Fanuc TP program (LS listing): CODE3.ls

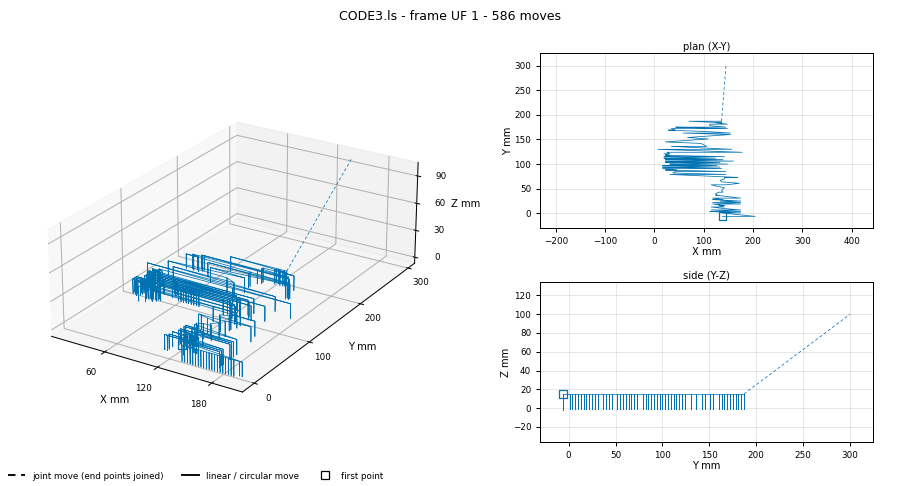
[picture p0: tool path of CODE3.ls in frame UF 1, 586 of 586 moves have a stored position in this frame; points joined in program order, loops and branches not executed]
/PROG CODE3
/ATTR
OWNER		= NOC_FANU;
COMMENT		= "NOC_FANUC";
PROG_SIZE	= 328;
CREATE		= DATE 97-07-08  TIME 03:05:20;
MODIFIED	= DATE 17-07-08  TIME 03:05:26;
FILE_NAME	= ;
VERSION		= 0;
LINE_COUNT	= 10;
MEMORY_SIZE	= 692;
PROTECT		= READ_WRITE;
TCD:  STACK_SIZE	= 0,
      TASK_PRIORITY	= 0,
      TIME_SLICE	= 0,
      BUSY_LAMP_OFF	= 0,
      ABORT_REQUEST	= 0,
      PAUSE_REQUEST	= 0;
DEFAULT_GROUP	= 1,*,*,*,*;
CONTROL_CODE	= 00000000 00000000;
/APPL
/MN
1:UFRAME_NUM=1 ;
2:UTOOL_NUM=3;
3:J P[133] 10% CNT100;
4:L P[134] 250mm/sec FINE;
5:L P[135] 250mm/sec CNT100;
6:L P[136] 250mm/sec CNT100;
7:L P[137] 250mm/sec FINE;
8:L P[138] 250mm/sec CNT100;
9:L P[139] 250mm/sec CNT100;
10:L P[140] 250mm/sec FINE;
11:L P[141] 250mm/sec CNT100;
12:L P[142] 250mm/sec CNT100;
13:L P[143] 250mm/sec FINE;
14:L P[144] 250mm/sec CNT100;
15:L P[145] 250mm/sec CNT100;
16:L P[146] 250mm/sec FINE;
17:L P[147] 250mm/sec CNT100;
18:L P[148] 250mm/sec CNT100;
19:L P[149] 250mm/sec FINE;
20:L P[150] 250mm/sec CNT100;
21:L P[151] 250mm/sec CNT100;
22:L P[152] 250mm/sec FINE;
23:L P[153] 250mm/sec CNT100;
24:L P[154] 250mm/sec CNT100;
25:L P[155] 250mm/sec FINE;
26:L P[156] 250mm/sec CNT100;
27:L P[157] 250mm/sec CNT100;
28:L P[158] 250mm/sec FINE;
29:L P[159] 250mm/sec CNT100;
30:L P[160] 250mm/sec CNT100;
31:L P[161] 250mm/sec FINE;
32:L P[162] 250mm/sec CNT100;
33:L P[163] 250mm/sec CNT100;
34:L P[164] 250mm/sec FINE;
35:L P[165] 250mm/sec CNT100;
36:L P[166] 250mm/sec CNT100;
37:L P[167] 250mm/sec FINE;
38:L P[168] 250mm/sec CNT100;
39:L P[169] 250mm/sec CNT100;
40:L P[170] 250mm/sec FINE;
41:L P[171] 250mm/sec CNT100;
42:L P[172] 250mm/sec CNT100;
43:L P[173] 250mm/sec FINE;
44:L P[174] 250mm/sec CNT100;
45:L P[175] 250mm/sec CNT100;
46:L P[176] 250mm/sec FINE;
47:L P[177] 250mm/sec CNT100;
48:L P[178] 250mm/sec CNT100;
49:L P[179] 250mm/sec FINE;
50:L P[180] 250mm/sec CNT100;
51:L P[181] 250mm/sec CNT100;
52:L P[182] 250mm/sec FINE;
53:L P[183] 250mm/sec CNT100;
54:L P[184] 250mm/sec CNT100;
55:L P[185] 250mm/sec FINE;
56:L P[186] 250mm/sec CNT100;
57:L P[187] 250mm/sec CNT100;
58:L P[188] 250mm/sec FINE;
59:L P[189] 250mm/sec CNT100;
60:L P[190] 250mm/sec CNT100;
61:L P[191] 250mm/sec FINE;
62:L P[192] 250mm/sec CNT100;
63:L P[193] 250mm/sec CNT100;
64:L P[194] 250mm/sec FINE;
65:L P[195] 250mm/sec CNT100;
66:L P[196] 250mm/sec CNT100;
67:L P[197] 250mm/sec FINE;
68:L P[198] 250mm/sec CNT100;
69:L P[532] 250mm/sec CNT100;
70:L P[533] 250mm/sec FINE;
71:L P[534] 250mm/sec CNT100;
72:L P[553] 250mm/sec CNT100;
73:L P[554] 250mm/sec FINE;
74:L P[555] 250mm/sec CNT100;
75:L P[670] 250mm/sec CNT100;
76:L P[671] 250mm/sec FINE;
77:L P[672] 250mm/sec CNT100;
78:L P[673] 250mm/sec CNT100;
79:L P[674] 250mm/sec FINE;
80:L P[675] 250mm/sec CNT100;
81:L P[691] 250mm/sec CNT100;
82:L P[692] 250mm/sec FINE;
83:L P[693] 250mm/sec CNT100;
84:L P[721] 250mm/sec CNT100;
85:L P[722] 250mm/sec FINE;
86:L P[723] 250mm/sec CNT100;
87:L P[841] 250mm/sec CNT100;
88:L P[842] 250mm/sec FINE;
89:L P[843] 250mm/sec CNT100;
90:L P[865] 250mm/sec CNT100;
91:L P[866] 250mm/sec FINE;
92:L P[867] 250mm/sec CNT100;
93:L P[880] 250mm/sec CNT100;
94:L P[881] 250mm/sec FINE;
95:L P[882] 250mm/sec CNT100;
96:L P[1024] 250mm/sec CNT100;
97:L P[1025] 250mm/sec FINE;
98:L P[1026] 250mm/sec CNT100;
99:L P[1162] 250mm/sec CNT100;
100:L P[1163] 250mm/sec FINE;
101:L P[1164] 250mm/sec CNT100;
102:L P[1186] 250mm/sec CNT100;
103:L P[1187] 250mm/sec FINE;
104:L P[1188] 250mm/sec CNT100;
105:L P[1189] 250mm/sec CNT100;
106:L P[1190] 250mm/sec FINE;
107:L P[1191] 250mm/sec CNT100;
108:L P[1333] 250mm/sec CNT100;
109:L P[1334] 250mm/sec FINE;
110:L P[1335] 250mm/sec CNT100;
111:L P[1336] 250mm/sec CNT100;
112:L P[1337] 250mm/sec FINE;
113:L P[1338] 250mm/sec CNT100;
114:L P[1339] 250mm/sec CNT100;
115:L P[1340] 250mm/sec FINE;
116:L P[1341] 250mm/sec CNT100;
117:L P[1345] 250mm/sec CNT100;
118:L P[1346] 250mm/sec FINE;
119:L P[1347] 250mm/sec CNT100;
120:L P[1477] 250mm/sec CNT100;
121:L P[1478] 250mm/sec FINE;
122:L P[1479] 250mm/sec CNT100;
123:L P[1480] 250mm/sec CNT100;
124:L P[1481] 250mm/sec FINE;
125:L P[1482] 250mm/sec CNT100;
126:L P[1489] 250mm/sec CNT100;
127:L P[1490] 250mm/sec FINE;
128:L P[1491] 250mm/sec CNT100;
129:L P[1492] 250mm/sec CNT100;
130:L P[1493] 250mm/sec FINE;
131:L P[1494] 250mm/sec CNT100;
132:L P[1507] 250mm/sec CNT100;
133:L P[1508] 250mm/sec FINE;
134:L P[1509] 250mm/sec CNT100;
135:L P[1627] 250mm/sec CNT100;
136:L P[1628] 250mm/sec FINE;
137:L P[1629] 250mm/sec CNT100;
138:L P[1633] 250mm/sec CNT100;
139:L P[1634] 250mm/sec FINE;
140:L P[1635] 250mm/sec CNT100;
141:L P[1654] 250mm/sec CNT100;
142:L P[1655] 250mm/sec FINE;
143:L P[1656] 250mm/sec CNT100;
144:L P[1789] 250mm/sec CNT100;
145:L P[1790] 250mm/sec FINE;
146:L P[1791] 250mm/sec CNT100;
147:L P[1798] 250mm/sec CNT100;
148:L P[1799] 250mm/sec FINE;
149:L P[1800] 250mm/sec CNT100;
150:L P[1918] 250mm/sec CNT100;
151:L P[1919] 250mm/sec FINE;
152:L P[1920] 250mm/sec CNT100;
153:L P[1927] 250mm/sec CNT100;
154:L P[1928] 250mm/sec FINE;
155:L P[1929] 250mm/sec CNT100;
156:L P[1930] 250mm/sec CNT100;
157:L P[1931] 250mm/sec FINE;
158:L P[1932] 250mm/sec CNT100;
159:L P[1939] 250mm/sec CNT100;
160:L P[1940] 250mm/sec FINE;
161:L P[1941] 250mm/sec CNT100;
162:L P[2065] 250mm/sec CNT100;
163:L P[2066] 250mm/sec FINE;
164:L P[2067] 250mm/sec CNT100;
165:L P[2095] 250mm/sec CNT100;
166:L P[2096] 250mm/sec FINE;
167:L P[2097] 250mm/sec CNT100;
168:L P[2371] 250mm/sec CNT100;
169:L P[2372] 250mm/sec FINE;
170:L P[2373] 250mm/sec CNT100;
171:L P[2374] 250mm/sec CNT100;
172:L P[2375] 250mm/sec FINE;
173:L P[2376] 250mm/sec CNT100;
174:L P[2512] 250mm/sec CNT100;
175:L P[2513] 250mm/sec FINE;
176:L P[2514] 250mm/sec CNT100;
177:L P[2656] 250mm/sec CNT100;
178:L P[2657] 250mm/sec FINE;
179:L P[2658] 250mm/sec CNT100;
180:L P[2665] 250mm/sec CNT100;
181:L P[2666] 250mm/sec FINE;
182:L P[2667] 250mm/sec CNT100;
183:L P[2803] 250mm/sec CNT100;
184:L P[2804] 250mm/sec FINE;
185:L P[2805] 250mm/sec CNT100;
186:L P[3121] 250mm/sec CNT100;
187:L P[3122] 250mm/sec FINE;
188:L P[3123] 250mm/sec CNT100;
189:L P[3256] 250mm/sec CNT100;
190:L P[3257] 250mm/sec FINE;
191:L P[3258] 250mm/sec CNT100;
192:L P[3394] 250mm/sec CNT100;
193:L P[3395] 250mm/sec FINE;
194:L P[3396] 250mm/sec CNT100;
195:L P[3397] 250mm/sec CNT100;
196:L P[3398] 250mm/sec FINE;
197:L P[3399] 250mm/sec CNT100;
198:L P[3412] 250mm/sec CNT100;
199:L P[3413] 250mm/sec FINE;
200:L P[3414] 250mm/sec CNT100;
201:L P[3562] 250mm/sec CNT100;
202:L P[3563] 250mm/sec FINE;
203:L P[3564] 250mm/sec CNT100;
204:L P[3697] 250mm/sec CNT100;
205:L P[3698] 250mm/sec FINE;
206:L P[3699] 250mm/sec CNT100;
207:L P[3832] 250mm/sec CNT100;
208:L P[3833] 250mm/sec FINE;
209:L P[3834] 250mm/sec CNT100;
210:L P[3979] 250mm/sec CNT100;
211:L P[3980] 250mm/sec FINE;
212:L P[3981] 250mm/sec CNT100;
213:L P[4114] 250mm/sec CNT100;
214:L P[4115] 250mm/sec FINE;
215:L P[4116] 250mm/sec CNT100;
216:L P[4123] 250mm/sec CNT100;
217:L P[4124] 250mm/sec FINE;
218:L P[4125] 250mm/sec CNT100;
219:L P[4288] 250mm/sec CNT100;
220:L P[4289] 250mm/sec FINE;
221:L P[4290] 250mm/sec CNT100;
222:L P[4366] 250mm/sec CNT100;
223:L P[4367] 250mm/sec FINE;
224:L P[4368] 250mm/sec CNT100;
225:L P[4384] 250mm/sec CNT100;
226:L P[4385] 250mm/sec FINE;
227:L P[4386] 250mm/sec CNT100;
228:L P[4432] 250mm/sec CNT100;
229:L P[4433] 250mm/sec FINE;
230:L P[4434] 250mm/sec CNT100;
231:L P[4585] 250mm/sec CNT100;
232:L P[4586] 250mm/sec FINE;
233:L P[4587] 250mm/sec CNT100;
234:L P[4669] 250mm/sec CNT100;
235:L P[4670] 250mm/sec FINE;
236:L P[4671] 250mm/sec CNT100;
237:L P[4675] 250mm/sec CNT100;
238:L P[4676] 250mm/sec FINE;
239:L P[4677] 250mm/sec CNT100;
240:L P[4717] 250mm/sec CNT100;
241:L P[4718] 250mm/sec FINE;
242:L P[4719] 250mm/sec CNT100;
243:L P[4729] 250mm/sec CNT100;
244:L P[4730] 250mm/sec FINE;
245:L P[4731] 250mm/sec CNT100;
246:L P[4732] 250mm/sec CNT100;
247:L P[4733] 250mm/sec FINE;
248:L P[4734] 250mm/sec CNT100;
249:L P[4735] 250mm/sec CNT100;
250:L P[4736] 250mm/sec FINE;
251:L P[4737] 250mm/sec CNT100;
252:L P[4741] 250mm/sec CNT100;
253:L P[4742] 250mm/sec FINE;
254:L P[4743] 250mm/sec CNT100;
255:L P[4855] 250mm/sec CNT100;
256:L P[4856] 250mm/sec FINE;
257:L P[4857] 250mm/sec CNT100;
258:L P[4858] 250mm/sec CNT100;
259:L P[4859] 250mm/sec FINE;
260:L P[4860] 250mm/sec CNT100;
261:L P[4861] 250mm/sec CNT100;
262:L P[4862] 250mm/sec FINE;
263:L P[4863] 250mm/sec CNT100;
264:L P[4864] 250mm/sec CNT100;
265:L P[4865] 250mm/sec FINE;
266:L P[4866] 250mm/sec CNT100;
267:L P[4870] 250mm/sec CNT100;
268:L P[4871] 250mm/sec FINE;
269:L P[4872] 250mm/sec CNT100;
270:L P[4873] 250mm/sec CNT100;
271:L P[4874] 250mm/sec FINE;
272:L P[4875] 250mm/sec CNT100;
273:L P[4876] 250mm/sec CNT100;
274:L P[4877] 250mm/sec FINE;
275:L P[4878] 250mm/sec CNT100;
276:L P[4879] 250mm/sec CNT100;
277:L P[4880] 250mm/sec FINE;
278:L P[4881] 250mm/sec CNT100;
279:L P[4882] 250mm/sec CNT100;
280:L P[4883] 250mm/sec FINE;
281:L P[4884] 250mm/sec CNT100;
282:L P[4885] 250mm/sec CNT100;
283:L P[4886] 250mm/sec FINE;
284:L P[4887] 250mm/sec CNT100;
285:L P[4888] 250mm/sec CNT100;
286:L P[4889] 250mm/sec FINE;
287:L P[4890] 250mm/sec CNT100;
288:L P[4963] 250mm/sec CNT100;
289:L P[4964] 250mm/sec FINE;
290:L P[4965] 250mm/sec CNT100;
291:L P[5002] 250mm/sec CNT100;
292:L P[5003] 250mm/sec FINE;
293:L P[5004] 250mm/sec CNT100;
294:L P[5005] 250mm/sec CNT100;
295:L P[5006] 250mm/sec FINE;
296:L P[5007] 250mm/sec CNT100;
297:L P[5011] 250mm/sec CNT100;
298:L P[5012] 250mm/sec FINE;
299:L P[5013] 250mm/sec CNT100;
300:L P[5032] 250mm/sec CNT100;
301:L P[5033] 250mm/sec FINE;
302:L P[5034] 250mm/sec CNT100;
303:L P[5095] 250mm/sec CNT100;
304:L P[5096] 250mm/sec FINE;
305:L P[5097] 250mm/sec CNT100;
306:L P[5098] 250mm/sec CNT100;
307:L P[5099] 250mm/sec FINE;
308:L P[5100] 250mm/sec CNT100;
309:L P[5143] 250mm/sec CNT100;
310:L P[5144] 250mm/sec FINE;
311:L P[5145] 250mm/sec CNT100;
312:L P[5149] 250mm/sec CNT100;
313:L P[5150] 250mm/sec FINE;
314:L P[5151] 250mm/sec CNT100;
315:L P[5152] 250mm/sec CNT100;
316:L P[5153] 250mm/sec FINE;
317:L P[5154] 250mm/sec CNT100;
318:L P[5245] 250mm/sec CNT100;
319:L P[5246] 250mm/sec FINE;
320:L P[5247] 250mm/sec CNT100;
321:L P[5254] 250mm/sec CNT100;
322:L P[5255] 250mm/sec FINE;
323:L P[5256] 250mm/sec CNT100;
324:L P[5326] 250mm/sec CNT100;
325:L P[5327] 250mm/sec FINE;
326:L P[5328] 250mm/sec CNT100;
327:L P[5329] 250mm/sec CNT100;
328:L P[5330] 250mm/sec FINE;
329:L P[5331] 250mm/sec CNT100;
330:L P[5332] 250mm/sec CNT100;
331:L P[5333] 250mm/sec FINE;
332:L P[5334] 250mm/sec CNT100;
333:L P[5359] 250mm/sec CNT100;
334:L P[5360] 250mm/sec FINE;
335:L P[5361] 250mm/sec CNT100;
336:L P[5362] 250mm/sec CNT100;
337:L P[5363] 250mm/sec FINE;
338:L P[5364] 250mm/sec CNT100;
339:L P[5365] 250mm/sec CNT100;
340:L P[5366] 250mm/sec FINE;
341:L P[5367] 250mm/sec CNT100;
342:L P[5368] 250mm/sec CNT100;
343:L P[5369] 250mm/sec FINE;
344:L P[5370] 250mm/sec CNT100;
345:L P[5371] 250mm/sec CNT100;
346:L P[5372] 250mm/sec FINE;
347:L P[5373] 250mm/sec CNT100;
348:L P[5374] 250mm/sec CNT100;
349:L P[5375] 250mm/sec FINE;
350:L P[5376] 250mm/sec CNT100;
351:L P[5377] 250mm/sec CNT100;
352:L P[5378] 250mm/sec FINE;
353:L P[5379] 250mm/sec CNT100;
354:L P[5380] 250mm/sec CNT100;
355:L P[5381] 250mm/sec FINE;
356:L P[5382] 250mm/sec CNT100;
357:L P[5383] 250mm/sec CNT100;
358:L P[5384] 250mm/sec FINE;
359:L P[5385] 250mm/sec CNT100;
360:L P[5416] 250mm/sec CNT100;
361:L P[5417] 250mm/sec FINE;
362:L P[5418] 250mm/sec CNT100;
363:L P[5419] 250mm/sec CNT100;
364:L P[5420] 250mm/sec FINE;
365:L P[5421] 250mm/sec CNT100;
366:L P[5440] 250mm/sec CNT100;
367:L P[5441] 250mm/sec FINE;
368:L P[5442] 250mm/sec CNT100;
369:L P[5443] 250mm/sec CNT100;
370:L P[5444] 250mm/sec FINE;
371:L P[5445] 250mm/sec CNT100;
372:L P[5485] 250mm/sec CNT100;
373:L P[5486] 250mm/sec FINE;
374:L P[5487] 250mm/sec CNT100;
375:L P[5488] 250mm/sec CNT100;
376:L P[5489] 250mm/sec FINE;
377:L P[5490] 250mm/sec CNT100;
378:L P[5518] 250mm/sec CNT100;
379:L P[5519] 250mm/sec FINE;
380:L P[5520] 250mm/sec CNT100;
381:L P[5596] 250mm/sec CNT100;
382:L P[5597] 250mm/sec FINE;
383:L P[5598] 250mm/sec CNT100;
384:L P[5656] 250mm/sec CNT100;
385:L P[5657] 250mm/sec FINE;
386:L P[5658] 250mm/sec CNT100;
387:L P[5662] 250mm/sec CNT100;
388:L P[5663] 250mm/sec FINE;
389:L P[5664] 250mm/sec CNT100;
390:L P[5665] 250mm/sec CNT100;
391:L P[5666] 250mm/sec FINE;
392:L P[5667] 250mm/sec CNT100;
393:L P[5677] 250mm/sec CNT100;
394:L P[5678] 250mm/sec FINE;
395:L P[5679] 250mm/sec CNT100;
396:L P[5734] 250mm/sec CNT100;
397:L P[5735] 250mm/sec FINE;
398:L P[5736] 250mm/sec CNT100;
399:L P[5740] 250mm/sec CNT100;
400:L P[5741] 250mm/sec FINE;
401:L P[5742] 250mm/sec CNT100;
402:L P[5779] 250mm/sec CNT100;
403:L P[5780] 250mm/sec FINE;
404:L P[5781] 250mm/sec CNT100;
405:L P[5782] 250mm/sec CNT100;
406:L P[5783] 250mm/sec FINE;
407:L P[5784] 250mm/sec CNT100;
408:L P[5785] 250mm/sec CNT100;
409:L P[5786] 250mm/sec FINE;
410:L P[5787] 250mm/sec CNT100;
411:L P[5812] 250mm/sec CNT100;
412:L P[5813] 250mm/sec FINE;
413:L P[5814] 250mm/sec CNT100;
414:L P[5833] 250mm/sec CNT100;
415:L P[5834] 250mm/sec FINE;
416:L P[5835] 250mm/sec CNT100;
417:L P[5836] 250mm/sec CNT100;
418:L P[5837] 250mm/sec FINE;
419:L P[5838] 250mm/sec CNT100;
420:L P[5845] 250mm/sec CNT100;
421:L P[5846] 250mm/sec FINE;
422:L P[5847] 250mm/sec CNT100;
423:L P[5881] 250mm/sec CNT100;
424:L P[5882] 250mm/sec FINE;
425:L P[5883] 250mm/sec CNT100;
426:L P[5884] 250mm/sec CNT100;
427:L P[5885] 250mm/sec FINE;
428:L P[5886] 250mm/sec CNT100;
429:L P[5914] 250mm/sec CNT100;
430:L P[5915] 250mm/sec FINE;
431:L P[5916] 250mm/sec CNT100;
432:L P[5917] 250mm/sec CNT100;
433:L P[5918] 250mm/sec FINE;
434:L P[5919] 250mm/sec CNT100;
435:L P[5929] 250mm/sec CNT100;
436:L P[5930] 250mm/sec FINE;
437:L P[5931] 250mm/sec CNT100;
438:L P[5968] 250mm/sec CNT100;
439:L P[5969] 250mm/sec FINE;
440:L P[5970] 250mm/sec CNT100;
441:L P[5971] 250mm/sec CNT100;
442:L P[5972] 250mm/sec FINE;
443:L P[5973] 250mm/sec CNT100;
444:L P[6034] 250mm/sec CNT100;
445:L P[6035] 250mm/sec FINE;
446:L P[6036] 250mm/sec CNT100;
447:L P[6064] 250mm/sec CNT100;
448:L P[6065] 250mm/sec FINE;
449:L P[6066] 250mm/sec CNT100;
450:L P[6073] 250mm/sec CNT100;
451:L P[6074] 250mm/sec FINE;
452:L P[6075] 250mm/sec CNT100;
453:L P[6163] 250mm/sec CNT100;
454:L P[6164] 250mm/sec FINE;
455:L P[6165] 250mm/sec CNT100;
456:L P[6166] 250mm/sec CNT100;
457:L P[6167] 250mm/sec FINE;
458:L P[6168] 250mm/sec CNT100;
459:L P[6169] 250mm/sec CNT100;
460:L P[6170] 250mm/sec FINE;
461:L P[6171] 250mm/sec CNT100;
462:L P[6175] 250mm/sec CNT100;
463:L P[6176] 250mm/sec FINE;
464:L P[6177] 250mm/sec CNT100;
465:L P[6280] 250mm/sec CNT100;
466:L P[6281] 250mm/sec FINE;
467:L P[6282] 250mm/sec CNT100;
468:L P[6325] 250mm/sec CNT100;
469:L P[6326] 250mm/sec FINE;
470:L P[6327] 250mm/sec CNT100;
471:L P[6376] 250mm/sec CNT100;
472:L P[6377] 250mm/sec FINE;
473:L P[6378] 250mm/sec CNT100;
474:L P[6496] 250mm/sec CNT100;
475:L P[6497] 250mm/sec FINE;
476:L P[6498] 250mm/sec CNT100;
477:L P[6601] 250mm/sec CNT100;
478:L P[6602] 250mm/sec FINE;
479:L P[6603] 250mm/sec CNT100;
480:L P[6745] 250mm/sec CNT100;
481:L P[6746] 250mm/sec FINE;
482:L P[6747] 250mm/sec CNT100;
483:L P[6778] 250mm/sec CNT100;
484:L P[6779] 250mm/sec FINE;
485:L P[6780] 250mm/sec CNT100;
486:L P[6988] 250mm/sec CNT100;
487:L P[6989] 250mm/sec FINE;
488:L P[6990] 250mm/sec CNT100;
489:L P[7054] 250mm/sec CNT100;
490:L P[7055] 250mm/sec FINE;
491:L P[7056] 250mm/sec CNT100;
492:L P[7312] 250mm/sec CNT100;
493:L P[7313] 250mm/sec FINE;
494:L P[7314] 250mm/sec CNT100;
495:L P[7414] 250mm/sec CNT100;
496:L P[7415] 250mm/sec FINE;
497:L P[7416] 250mm/sec CNT100;
498:L P[7657] 250mm/sec CNT100;
499:L P[7658] 250mm/sec FINE;
500:L P[7659] 250mm/sec CNT100;
501:L P[7660] 250mm/sec CNT100;
502:L P[7661] 250mm/sec FINE;
503:L P[7662] 250mm/sec CNT100;
504:L P[7699] 250mm/sec CNT100;
505:L P[7700] 250mm/sec FINE;
506:L P[7701] 250mm/sec CNT100;
507:L P[7705] 250mm/sec CNT100;
508:L P[7706] 250mm/sec FINE;
509:L P[7707] 250mm/sec CNT100;
510:L P[7750] 250mm/sec CNT100;
511:L P[7751] 250mm/sec FINE;
512:L P[7752] 250mm/sec CNT100;
513:L P[7753] 250mm/sec CNT100;
514:L P[7754] 250mm/sec FINE;
515:L P[7755] 250mm/sec CNT100;
516:L P[7792] 250mm/sec CNT100;
517:L P[7793] 250mm/sec FINE;
518:L P[7794] 250mm/sec CNT100;
519:L P[7843] 250mm/sec CNT100;
520:L P[7844] 250mm/sec FINE;
521:L P[7845] 250mm/sec CNT100;
522:L P[7852] 250mm/sec CNT100;
523:L P[7853] 250mm/sec FINE;
524:L P[7854] 250mm/sec CNT100;
525:L P[7858] 250mm/sec CNT100;
526:L P[7859] 250mm/sec FINE;
527:L P[7860] 250mm/sec CNT100;
528:L P[7927] 250mm/sec CNT100;
529:L P[7928] 250mm/sec FINE;
530:L P[7929] 250mm/sec CNT100;
531:L P[7930] 250mm/sec CNT100;
532:L P[7931] 250mm/sec FINE;
533:L P[7932] 250mm/sec CNT100;
534:L P[7936] 250mm/sec CNT100;
535:L P[7937] 250mm/sec FINE;
536:L P[7938] 250mm/sec CNT100;
537:L P[7987] 250mm/sec CNT100;
538:L P[7988] 250mm/sec FINE;
539:L P[7989] 250mm/sec CNT100;
540:L P[8002] 250mm/sec CNT100;
541:L P[8003] 250mm/sec FINE;
542:L P[8004] 250mm/sec CNT100;
543:L P[8005] 250mm/sec CNT100;
544:L P[8006] 250mm/sec FINE;
545:L P[8007] 250mm/sec CNT100;
546:L P[8011] 250mm/sec CNT100;
547:L P[8012] 250mm/sec FINE;
548:L P[8013] 250mm/sec CNT100;
549:L P[8047] 250mm/sec CNT100;
550:L P[8048] 250mm/sec FINE;
551:L P[8049] 250mm/sec CNT100;
552:L P[8077] 250mm/sec CNT100;
553:L P[8078] 250mm/sec FINE;
554:L P[8079] 250mm/sec CNT100;
555:L P[8161] 250mm/sec CNT100;
556:L P[8162] 250mm/sec FINE;
557:L P[8163] 250mm/sec CNT100;
558:L P[8197] 250mm/sec CNT100;
559:L P[8198] 250mm/sec FINE;
560:L P[8199] 250mm/sec CNT100;
561:L P[8275] 250mm/sec CNT100;
562:L P[8276] 250mm/sec FINE;
563:L P[8277] 250mm/sec CNT100;
564:L P[8281] 250mm/sec CNT100;
565:L P[8282] 250mm/sec FINE;
566:L P[8283] 250mm/sec CNT100;
567:L P[8284] 250mm/sec CNT100;
568:L P[8285] 250mm/sec FINE;
569:L P[8286] 250mm/sec CNT100;
570:L P[8287] 250mm/sec CNT100;
571:L P[8288] 250mm/sec FINE;
572:L P[8289] 250mm/sec CNT100;
573:L P[8398] 250mm/sec CNT100;
574:L P[8399] 250mm/sec FINE;
575:L P[8400] 250mm/sec CNT100;
576:L P[8452] 250mm/sec CNT100;
577:L P[8453] 250mm/sec FINE;
578:L P[8454] 250mm/sec CNT100;
579:L P[8455] 250mm/sec CNT100;
580:L P[8456] 250mm/sec FINE;
581:L P[8457] 250mm/sec CNT100;
582:L P[8461] 250mm/sec CNT100;
583:L P[8462] 250mm/sec FINE;
584:L P[8463] 250mm/sec CNT100;
585:L P[8464] 250mm/sec CNT100;
586:L P[8465] 250mm/sec FINE;
587:L P[8466] 250mm/sec CNT100;
588:J P[11569] 50% CNT100;
/POS
P[133]{
   GP1:
	UF : 1, UT : 3,		CONFIG : 'N U T, 0, 0, 0',
	X =  138.000  mm,	Y =  -6.000  mm,	Z =   15.000 mm,
	W =-180.000 deg,	P =   0.000 deg,	R =    90.000 deg
};
P[134]{
   GP1:
	UF : 1, UT : 3,		CONFIG : 'N U T, 0, 0, 0',
	X =  138.000  mm,	Y =  -6.000  mm,	Z =   -2.000 mm,
	W =-180.000 deg,	P =   0.000 deg,	R =    90.000 deg
};
P[135]{
   GP1:
	UF : 1, UT : 3,		CONFIG : 'N U T, 0, 0, 0',
	X =  138.000  mm,	Y =  -6.000  mm,	Z =   15.000 mm,
	W =-180.000 deg,	P =   0.000 deg,	R =    90.000 deg
};
P[136]{
   GP1:
	UF : 1, UT : 3,		CONFIG : 'N U T, 0, 0, 0',
	X =  141.000  mm,	Y =  -6.000  mm,	Z =   15.000 mm,
	W =-180.000 deg,	P =   0.000 deg,	R =    90.000 deg
};
P[137]{
   GP1:
	UF : 1, UT : 3,		CONFIG : 'N U T, 0, 0, 0',
	X =  141.000  mm,	Y =  -6.000  mm,	Z =   -2.000 mm,
	W =-180.000 deg,	P =   0.000 deg,	R =    90.000 deg
};
P[138]{
   GP1:
	UF : 1, UT : 3,		CONFIG : 'N U T, 0, 0, 0',
	X =  141.000  mm,	Y =  -6.000  mm,	Z =   15.000 mm,
	W =-180.000 deg,	P =   0.000 deg,	R =    90.000 deg
};
P[139]{
   GP1:
	UF : 1, UT : 3,		CONFIG : 'N U T, 0, 0, 0',
	X =  144.000  mm,	Y =  -6.000  mm,	Z =   15.000 mm,
	W =-180.000 deg,	P =   0.000 deg,	R =    90.000 deg
};
P[140]{
   GP1:
	UF : 1, UT : 3,		CONFIG : 'N U T, 0, 0, 0',
	X =  144.000  mm,	Y =  -6.000  mm,	Z =   -2.000 mm,
	W =-180.000 deg,	P =   0.000 deg,	R =    90.000 deg
};
P[141]{
   GP1:
	UF : 1, UT : 3,		CONFIG : 'N U T, 0, 0, 0',
	X =  144.000  mm,	Y =  -6.000  mm,	Z =   15.000 mm,
	W =-180.000 deg,	P =   0.000 deg,	R =    90.000 deg
};
P[142]{
   GP1:
	UF : 1, UT : 3,		CONFIG : 'N U T, 0, 0, 0',
	X =  147.000  mm,	Y =  -6.000  mm,	Z =   15.000 mm,
	W =-180.000 deg,	P =   0.000 deg,	R =    90.000 deg
};
P[143]{
   GP1:
	UF : 1, UT : 3,		CONFIG : 'N U T, 0, 0, 0',
	X =  147.000  mm,	Y =  -6.000  mm,	Z =   -2.000 mm,
	W =-180.000 deg,	P =   0.000 deg,	R =    90.000 deg
};
P[144]{
   GP1:
	UF : 1, UT : 3,		CONFIG : 'N U T, 0, 0, 0',
	X =  147.000  mm,	Y =  -6.000  mm,	Z =   15.000 mm,
	W =-180.000 deg,	P =   0.000 deg,	R =    90.000 deg
};
P[145]{
   GP1:
	UF : 1, UT : 3,		CONFIG : 'N U T, 0, 0, 0',
	X =  150.000  mm,	Y =  -6.000  mm,	Z =   15.000 mm,
	W =-180.000 deg,	P =   0.000 deg,	R =    90.000 deg
};
P[146]{
   GP1:
	UF : 1, UT : 3,		CONFIG : 'N U T, 0, 0, 0',
	X =  150.000  mm,	Y =  -6.000  mm,	Z =   -2.000 mm,
	W =-180.000 deg,	P =   0.000 deg,	R =    90.000 deg
};
P[147]{
   GP1:
	UF : 1, UT : 3,		CONFIG : 'N U T, 0, 0, 0',
	X =  150.000  mm,	Y =  -6.000  mm,	Z =   15.000 mm,
	W =-180.000 deg,	P =   0.000 deg,	R =    90.000 deg
};
P[148]{
   GP1:
	UF : 1, UT : 3,		CONFIG : 'N U T, 0, 0, 0',
	X =  153.000  mm,	Y =  -6.000  mm,	Z =   15.000 mm,
	W =-180.000 deg,	P =   0.000 deg,	R =    90.000 deg
};
P[149]{
   GP1:
	UF : 1, UT : 3,		CONFIG : 'N U T, 0, 0, 0',
	X =  153.000  mm,	Y =  -6.000  mm,	Z =   -2.000 mm,
	W =-180.000 deg,	P =   0.000 deg,	R =    90.000 deg
};
P[150]{
   GP1:
	UF : 1, UT : 3,		CONFIG : 'N U T, 0, 0, 0',
	X =  153.000  mm,	Y =  -6.000  mm,	Z =   15.000 mm,
	W =-180.000 deg,	P =   0.000 deg,	R =    90.000 deg
};
P[151]{
   GP1:
	UF : 1, UT : 3,		CONFIG : 'N U T, 0, 0, 0',
	X =  156.000  mm,	Y =  -6.000  mm,	Z =   15.000 mm,
	W =-180.000 deg,	P =   0.000 deg,	R =    90.000 deg
};
P[152]{
   GP1:
	UF : 1, UT : 3,		CONFIG : 'N U T, 0, 0, 0',
	X =  156.000  mm,	Y =  -6.000  mm,	Z =   -2.000 mm,
	W =-180.000 deg,	P =   0.000 deg,	R =    90.000 deg
};
P[153]{
   GP1:
	UF : 1, UT : 3,		CONFIG : 'N U T, 0, 0, 0',
	X =  156.000  mm,	Y =  -6.000  mm,	Z =   15.000 mm,
	W =-180.000 deg,	P =   0.000 deg,	R =    90.000 deg
};
P[154]{
   GP1:
	UF : 1, UT : 3,		CONFIG : 'N U T, 0, 0, 0',
	X =  159.000  mm,	Y =  -6.000  mm,	Z =   15.000 mm,
	W =-180.000 deg,	P =   0.000 deg,	R =    90.000 deg
};
P[155]{
   GP1:
	UF : 1, UT : 3,		CONFIG : 'N U T, 0, 0, 0',
	X =  159.000  mm,	Y =  -6.000  mm,	Z =   -2.000 mm,
	W =-180.000 deg,	P =   0.000 deg,	R =    90.000 deg
};
P[156]{
   GP1:
	UF : 1, UT : 3,		CONFIG : 'N U T, 0, 0, 0',
	X =  159.000  mm,	Y =  -6.000  mm,	Z =   15.000 mm,
	W =-180.000 deg,	P =   0.000 deg,	R =    90.000 deg
};
P[157]{
   GP1:
	UF : 1, UT : 3,		CONFIG : 'N U T, 0, 0, 0',
	X =  162.000  mm,	Y =  -6.000  mm,	Z =   15.000 mm,
	W =-180.000 deg,	P =   0.000 deg,	R =    90.000 deg
};
P[158]{
   GP1:
	UF : 1, UT : 3,		CONFIG : 'N U T, 0, 0, 0',
	X =  162.000  mm,	Y =  -6.000  mm,	Z =   -2.000 mm,
	W =-180.000 deg,	P =   0.000 deg,	R =    90.000 deg
};
P[159]{
   GP1:
	UF : 1, UT : 3,		CONFIG : 'N U T, 0, 0, 0',
	X =  162.000  mm,	Y =  -6.000  mm,	Z =   15.000 mm,
	W =-180.000 deg,	P =   0.000 deg,	R =    90.000 deg
};
P[160]{
   GP1:
	UF : 1, UT : 3,		CONFIG : 'N U T, 0, 0, 0',
	X =  165.000  mm,	Y =  -6.000  mm,	Z =   15.000 mm,
	W =-180.000 deg,	P =   0.000 deg,	R =    90.000 deg
};
P[161]{
   GP1:
	UF : 1, UT : 3,		CONFIG : 'N U T, 0, 0, 0',
	X =  165.000  mm,	Y =  -6.000  mm,	Z =   -2.000 mm,
	W =-180.000 deg,	P =   0.000 deg,	R =    90.000 deg
};
P[162]{
   GP1:
	UF : 1, UT : 3,		CONFIG : 'N U T, 0, 0, 0',
	X =  165.000  mm,	Y =  -6.000  mm,	Z =   15.000 mm,
	W =-180.000 deg,	P =   0.000 deg,	R =    90.000 deg
};
P[163]{
   GP1:
	UF : 1, UT : 3,		CONFIG : 'N U T, 0, 0, 0',
	X =  168.000  mm,	Y =  -6.000  mm,	Z =   15.000 mm,
	W =-180.000 deg,	P =   0.000 deg,	R =    90.000 deg
};
P[164]{
   GP1:
	UF : 1, UT : 3,		CONFIG : 'N U T, 0, 0, 0',
	X =  168.000  mm,	Y =  -6.000  mm,	Z =   -2.000 mm,
	W =-180.000 deg,	P =   0.000 deg,	R =    90.000 deg
};
P[165]{
   GP1:
	UF : 1, UT : 3,		CONFIG : 'N U T, 0, 0, 0',
	X =  168.000  mm,	Y =  -6.000  mm,	Z =   15.000 mm,
	W =-180.000 deg,	P =   0.000 deg,	R =    90.000 deg
};
P[166]{
   GP1:
	UF : 1, UT : 3,		CONFIG : 'N U T, 0, 0, 0',
	X =  171.000  mm,	Y =  -6.000  mm,	Z =   15.000 mm,
	W =-180.000 deg,	P =   0.000 deg,	R =    90.000 deg
};
P[167]{
   GP1:
	UF : 1, UT : 3,		CONFIG : 'N U T, 0, 0, 0',
	X =  171.000  mm,	Y =  -6.000  mm,	Z =   -2.000 mm,
	W =-180.000 deg,	P =   0.000 deg,	R =    90.000 deg
};
P[168]{
   GP1:
	UF : 1, UT : 3,		CONFIG : 'N U T, 0, 0, 0',
	X =  171.000  mm,	Y =  -6.000  mm,	Z =   15.000 mm,
	W =-180.000 deg,	P =   0.000 deg,	R =    90.000 deg
};
P[169]{
   GP1:
	UF : 1, UT : 3,		CONFIG : 'N U T, 0, 0, 0',
	X =  174.000  mm,	Y =  -6.000  mm,	Z =   15.000 mm,
	W =-180.000 deg,	P =   0.000 deg,	R =    90.000 deg
};
P[170]{
   GP1:
	UF : 1, UT : 3,		CONFIG : 'N U T, 0, 0, 0',
	X =  174.000  mm,	Y =  -6.000  mm,	Z =   -2.000 mm,
	W =-180.000 deg,	P =   0.000 deg,	R =    90.000 deg
};
P[171]{
   GP1:
	UF : 1, UT : 3,		CONFIG : 'N U T, 0, 0, 0',
	X =  174.000  mm,	Y =  -6.000  mm,	Z =   15.000 mm,
	W =-180.000 deg,	P =   0.000 deg,	R =    90.000 deg
};
P[172]{
   GP1:
	UF : 1, UT : 3,		CONFIG : 'N U T, 0, 0, 0',
	X =  177.000  mm,	Y =  -6.000  mm,	Z =   15.000 mm,
	W =-180.000 deg,	P =   0.000 deg,	R =    90.000 deg
};
P[173]{
   GP1:
	UF : 1, UT : 3,		CONFIG : 'N U T, 0, 0, 0',
	X =  177.000  mm,	Y =  -6.000  mm,	Z =   -2.000 mm,
	W =-180.000 deg,	P =   0.000 deg,	R =    90.000 deg
};
P[174]{
   GP1:
	UF : 1, UT : 3,		CONFIG : 'N U T, 0, 0, 0',
	X =  177.000  mm,	Y =  -6.000  mm,	Z =   15.000 mm,
	W =-180.000 deg,	P =   0.000 deg,	R =    90.000 deg
};
P[175]{
   GP1:
	UF : 1, UT : 3,		CONFIG : 'N U T, 0, 0, 0',
	X =  180.000  mm,	Y =  -6.000  mm,	Z =   15.000 mm,
	W =-180.000 deg,	P =   0.000 deg,	R =    90.000 deg
};
P[176]{
   GP1:
	UF : 1, UT : 3,		CONFIG : 'N U T, 0, 0, 0',
	X =  180.000  mm,	Y =  -6.000  mm,	Z =   -2.000 mm,
	W =-180.000 deg,	P =   0.000 deg,	R =    90.000 deg
};
P[177]{
   GP1:
	UF : 1, UT : 3,		CONFIG : 'N U T, 0, 0, 0',
	X =  180.000  mm,	Y =  -6.000  mm,	Z =   15.000 mm,
	W =-180.000 deg,	P =   0.000 deg,	R =    90.000 deg
};
P[178]{
   GP1:
	UF : 1, UT : 3,		CONFIG : 'N U T, 0, 0, 0',
	X =  183.000  mm,	Y =  -6.000  mm,	Z =   15.000 mm,
	W =-180.000 deg,	P =   0.000 deg,	R =    90.000 deg
};
P[179]{
   GP1:
	UF : 1, UT : 3,		CONFIG : 'N U T, 0, 0, 0',
	X =  183.000  mm,	Y =  -6.000  mm,	Z =   -2.000 mm,
	W =-180.000 deg,	P =   0.000 deg,	R =    90.000 deg
};
P[180]{
   GP1:
	UF : 1, UT : 3,		CONFIG : 'N U T, 0, 0, 0',
	X =  183.000  mm,	Y =  -6.000  mm,	Z =   15.000 mm,
	W =-180.000 deg,	P =   0.000 deg,	R =    90.000 deg
};
P[181]{
   GP1:
	UF : 1, UT : 3,		CONFIG : 'N U T, 0, 0, 0',
	X =  186.000  mm,	Y =  -6.000  mm,	Z =   15.000 mm,
	W =-180.000 deg,	P =   0.000 deg,	R =    90.000 deg
};
P[182]{
   GP1:
	UF : 1, UT : 3,		CONFIG : 'N U T, 0, 0, 0',
	X =  186.000  mm,	Y =  -6.000  mm,	Z =   -2.000 mm,
	W =-180.000 deg,	P =   0.000 deg,	R =    90.000 deg
};
P[183]{
   GP1:
	UF : 1, UT : 3,		CONFIG : 'N U T, 0, 0, 0',
	X =  186.000  mm,	Y =  -6.000  mm,	Z =   15.000 mm,
	W =-180.000 deg,	P =   0.000 deg,	R =    90.000 deg
};
P[184]{
   GP1:
	UF : 1, UT : 3,		CONFIG : 'N U T, 0, 0, 0',
	X =  189.000  mm,	Y =  -6.000  mm,	Z =   15.000 mm,
	W =-180.000 deg,	P =   0.000 deg,	R =    90.000 deg
};
P[185]{
   GP1:
	UF : 1, UT : 3,		CONFIG : 'N U T, 0, 0, 0',
	X =  189.000  mm,	Y =  -6.000  mm,	Z =   -2.000 mm,
	W =-180.000 deg,	P =   0.000 deg,	R =    90.000 deg
};
P[186]{
   GP1:
	UF : 1, UT : 3,		CONFIG : 'N U T, 0, 0, 0',
	X =  189.000  mm,	Y =  -6.000  mm,	Z =   15.000 mm,
	W =-180.000 deg,	P =   0.000 deg,	R =    90.000 deg
};
P[187]{
   GP1:
	UF : 1, UT : 3,		CONFIG : 'N U T, 0, 0, 0',
	X =  192.000  mm,	Y =  -6.000  mm,	Z =   15.000 mm,
	W =-180.000 deg,	P =   0.000 deg,	R =    90.000 deg
};
P[188]{
   GP1:
	UF : 1, UT : 3,		CONFIG : 'N U T, 0, 0, 0',
	X =  192.000  mm,	Y =  -6.000  mm,	Z =   -2.000 mm,
	W =-180.000 deg,	P =   0.000 deg,	R =    90.000 deg
};
P[189]{
   GP1:
	UF : 1, UT : 3,		CONFIG : 'N U T, 0, 0, 0',
	X =  192.000  mm,	Y =  -6.000  mm,	Z =   15.000 mm,
	W =-180.000 deg,	P =   0.000 deg,	R =    90.000 deg
};
P[190]{
   GP1:
	UF : 1, UT : 3,		CONFIG : 'N U T, 0, 0, 0',
	X =  195.000  mm,	Y =  -6.000  mm,	Z =   15.000 mm,
	W =-180.000 deg,	P =   0.000 deg,	R =    90.000 deg
};
P[191]{
   GP1:
	UF : 1, UT : 3,		CONFIG : 'N U T, 0, 0, 0',
	X =  195.000  mm,	Y =  -6.000  mm,	Z =   -2.000 mm,
	W =-180.000 deg,	P =   0.000 deg,	R =    90.000 deg
};
P[192]{
   GP1:
	UF : 1, UT : 3,		CONFIG : 'N U T, 0, 0, 0',
	X =  195.000  mm,	Y =  -6.000  mm,	Z =   15.000 mm,
	W =-180.000 deg,	P =   0.000 deg,	R =    90.000 deg
};
P[193]{
   GP1:
	UF : 1, UT : 3,		CONFIG : 'N U T, 0, 0, 0',
	X =  201.000  mm,	Y =  -6.000  mm,	Z =   15.000 mm,
	W =-180.000 deg,	P =   0.000 deg,	R =    90.000 deg
};
P[194]{
   GP1:
	UF : 1, UT : 3,		CONFIG : 'N U T, 0, 0, 0',
	X =  201.000  mm,	Y =  -6.000  mm,	Z =   0.000 mm,
	W =-180.000 deg,	P =   0.000 deg,	R =    90.000 deg
};
P[195]{
   GP1:
	UF : 1, UT : 3,		CONFIG : 'N U T, 0, 0, 0',
	X =  201.000  mm,	Y =  -6.000  mm,	Z =   15.000 mm,
	W =-180.000 deg,	P =   0.000 deg,	R =    90.000 deg
};
P[196]{
   GP1:
	UF : 1, UT : 3,		CONFIG : 'N U T, 0, 0, 0',
	X =  204.000  mm,	Y =  -6.000  mm,	Z =   15.000 mm,
	W =-180.000 deg,	P =   0.000 deg,	R =    90.000 deg
};
P[197]{
   GP1:
	UF : 1, UT : 3,		CONFIG : 'N U T, 0, 0, 0',
	X =  204.000  mm,	Y =  -6.000  mm,	Z =   0.000 mm,
	W =-180.000 deg,	P =   0.000 deg,	R =    90.000 deg
};
P[198]{
   GP1:
	UF : 1, UT : 3,		CONFIG : 'N U T, 0, 0, 0',
	X =  204.000  mm,	Y =  -6.000  mm,	Z =   15.000 mm,
	W =-180.000 deg,	P =   0.000 deg,	R =    90.000 deg
};
P[532]{
   GP1:
	UF : 1, UT : 3,		CONFIG : 'N U T, 0, 0, 0',
	X =  136.000  mm,	Y =  1.000  mm,	Z =   15.000 mm,
	W =-180.000 deg,	P =   0.000 deg,	R =    90.000 deg
};
P[533]{
   GP1:
	UF : 1, UT : 3,		CONFIG : 'N U T, 0, 0, 0',
	X =  136.000  mm,	Y =  1.000  mm,	Z =   -1.000 mm,
	W =-180.000 deg,	P =   0.000 deg,	R =    90.000 deg
};
P[534]{
   GP1:
	UF : 1, UT : 3,		CONFIG : 'N U T, 0, 0, 0',
	X =  136.000  mm,	Y =  1.000  mm,	Z =   15.000 mm,
	W =-180.000 deg,	P =   0.000 deg,	R =    90.000 deg
};
P[553]{
   GP1:
	UF : 1, UT : 3,		CONFIG : 'N U T, 0, 0, 0',
	X =  175.000  mm,	Y =  1.000  mm,	Z =   15.000 mm,
	W =-180.000 deg,	P =   0.000 deg,	R =    90.000 deg
};
P[554]{
   GP1:
	UF : 1, UT : 3,		CONFIG : 'N U T, 0, 0, 0',
	X =  175.000  mm,	Y =  1.000  mm,	Z =   -1.000 mm,
	W =-180.000 deg,	P =   0.000 deg,	R =    90.000 deg
};
P[555]{
   GP1:
	UF : 1, UT : 3,		CONFIG : 'N U T, 0, 0, 0',
	X =  175.000  mm,	Y =  1.000  mm,	Z =   15.000 mm,
	W =-180.000 deg,	P =   0.000 deg,	R =    90.000 deg
};
P[670]{
   GP1:
	UF : 1, UT : 3,		CONFIG : 'N U T, 0, 0, 0',
	X =  112.000  mm,	Y =  4.000  mm,	Z =   15.000 mm,
	W =-180.000 deg,	P =   0.000 deg,	R =    90.000 deg
};
P[671]{
   GP1:
	UF : 1, UT : 3,		CONFIG : 'N U T, 0, 0, 0',
	X =  112.000  mm,	Y =  4.000  mm,	Z =   -1.000 mm,
	W =-180.000 deg,	P =   0.000 deg,	R =    90.000 deg
};
P[672]{
   GP1:
	UF : 1, UT : 3,		CONFIG : 'N U T, 0, 0, 0',
	X =  112.000  mm,	Y =  4.000  mm,	Z =   15.000 mm,
	W =-180.000 deg,	P =   0.000 deg,	R =    90.000 deg
};
P[673]{
   GP1:
	UF : 1, UT : 3,		CONFIG : 'N U T, 0, 0, 0',
	X =  115.000  mm,	Y =  4.000  mm,	Z =   15.000 mm,
	W =-180.000 deg,	P =   0.000 deg,	R =    90.000 deg
};
P[674]{
   GP1:
	UF : 1, UT : 3,		CONFIG : 'N U T, 0, 0, 0',
	X =  115.000  mm,	Y =  4.000  mm,	Z =   -1.000 mm,
	W =-180.000 deg,	P =   0.000 deg,	R =    90.000 deg
};
P[675]{
   GP1:
	UF : 1, UT : 3,		CONFIG : 'N U T, 0, 0, 0',
	X =  115.000  mm,	Y =  4.000  mm,	Z =   15.000 mm,
	W =-180.000 deg,	P =   0.000 deg,	R =    90.000 deg
};
P[691]{
   GP1:
	UF : 1, UT : 3,		CONFIG : 'N U T, 0, 0, 0',
	X =  133.000  mm,	Y =  4.000  mm,	Z =   15.000 mm,
	W =-180.000 deg,	P =   0.000 deg,	R =    90.000 deg
};
P[692]{
   GP1:
	UF : 1, UT : 3,		CONFIG : 'N U T, 0, 0, 0',
	X =  133.000  mm,	Y =  4.000  mm,	Z =   -1.000 mm,
	W =-180.000 deg,	P =   0.000 deg,	R =    90.000 deg
};
P[693]{
   GP1:
	UF : 1, UT : 3,		CONFIG : 'N U T, 0, 0, 0',
	X =  133.000  mm,	Y =  4.000  mm,	Z =   15.000 mm,
	W =-180.000 deg,	P =   0.000 deg,	R =    90.000 deg
};
P[721]{
   GP1:
	UF : 1, UT : 3,		CONFIG : 'N U T, 0, 0, 0',
	X =  175.000  mm,	Y =  4.000  mm,	Z =   15.000 mm,
	W =-180.000 deg,	P =   0.000 deg,	R =    90.000 deg
};
P[722]{
   GP1:
	UF : 1, UT : 3,		CONFIG : 'N U T, 0, 0, 0',
	X =  175.000  mm,	Y =  4.000  mm,	Z =   -1.000 mm,
	W =-180.000 deg,	P =   0.000 deg,	R =    90.000 deg
};
P[723]{
   GP1:
	UF : 1, UT : 3,		CONFIG : 'N U T, 0, 0, 0',
	X =  175.000  mm,	Y =  4.000  mm,	Z =   15.000 mm,
	W =-180.000 deg,	P =   0.000 deg,	R =    90.000 deg
};
P[841]{
   GP1:
	UF : 1, UT : 3,		CONFIG : 'N U T, 0, 0, 0',
	X =  115.000  mm,	Y =  7.000  mm,	Z =   15.000 mm,
	W =-180.000 deg,	P =   0.000 deg,	R =    90.000 deg
};
P[842]{
   GP1:
	UF : 1, UT : 3,		CONFIG : 'N U T, 0, 0, 0',
	X =  115.000  mm,	Y =  7.000  mm,	Z =   -1.000 mm,
	W =-180.000 deg,	P =   0.000 deg,	R =    90.000 deg
};
P[843]{
   GP1:
	UF : 1, UT : 3,		CONFIG : 'N U T, 0, 0, 0',
	X =  115.000  mm,	Y =  7.000  mm,	Z =   15.000 mm,
	W =-180.000 deg,	P =   0.000 deg,	R =    90.000 deg
};
P[865]{
   GP1:
	UF : 1, UT : 3,		CONFIG : 'N U T, 0, 0, 0',
	X =  139.000  mm,	Y =  7.000  mm,	Z =   15.000 mm,
	W =-180.000 deg,	P =   0.000 deg,	R =    90.000 deg
};
P[866]{
   GP1:
	UF : 1, UT : 3,		CONFIG : 'N U T, 0, 0, 0',
	X =  139.000  mm,	Y =  7.000  mm,	Z =   -1.000 mm,
	W =-180.000 deg,	P =   0.000 deg,	R =    90.000 deg
};
P[867]{
   GP1:
	UF : 1, UT : 3,		CONFIG : 'N U T, 0, 0, 0',
	X =  139.000  mm,	Y =  7.000  mm,	Z =   15.000 mm,
	W =-180.000 deg,	P =   0.000 deg,	R =    90.000 deg
};
P[880]{
   GP1:
	UF : 1, UT : 3,		CONFIG : 'N U T, 0, 0, 0',
	X =  175.000  mm,	Y =  7.000  mm,	Z =   15.000 mm,
	W =-180.000 deg,	P =   0.000 deg,	R =    90.000 deg
};
P[881]{
   GP1:
	UF : 1, UT : 3,		CONFIG : 'N U T, 0, 0, 0',
	X =  175.000  mm,	Y =  7.000  mm,	Z =   -1.000 mm,
	W =-180.000 deg,	P =   0.000 deg,	R =    90.000 deg
};
P[882]{
   GP1:
	UF : 1, UT : 3,		CONFIG : 'N U T, 0, 0, 0',
	X =  175.000  mm,	Y =  7.000  mm,	Z =   15.000 mm,
	W =-180.000 deg,	P =   0.000 deg,	R =    90.000 deg
};
P[1024]{
   GP1:
	UF : 1, UT : 3,		CONFIG : 'N U T, 0, 0, 0',
	X =  139.000  mm,	Y =  10.000  mm,	Z =   15.000 mm,
	W =-180.000 deg,	P =   0.000 deg,	R =    90.000 deg
};
P[1025]{
   GP1:
	UF : 1, UT : 3,		CONFIG : 'N U T, 0, 0, 0',
	X =  139.000  mm,	Y =  10.000  mm,	Z =   -1.000 mm,
	W =-180.000 deg,	P =   0.000 deg,	R =    90.000 deg
};
P[1026]{
   GP1:
	UF : 1, UT : 3,		CONFIG : 'N U T, 0, 0, 0',
	X =  139.000  mm,	Y =  10.000  mm,	Z =   15.000 mm,
	W =-180.000 deg,	P =   0.000 deg,	R =    90.000 deg
};
P[1162]{
   GP1:
	UF : 1, UT : 3,		CONFIG : 'N U T, 0, 0, 0',
	X =  115.000  mm,	Y =  13.000  mm,	Z =   15.000 mm,
	W =-180.000 deg,	P =   0.000 deg,	R =    90.000 deg
};
P[1163]{
   GP1:
	UF : 1, UT : 3,		CONFIG : 'N U T, 0, 0, 0',
	X =  115.000  mm,	Y =  13.000  mm,	Z =   -1.000 mm,
	W =-180.000 deg,	P =   0.000 deg,	R =    90.000 deg
};
P[1164]{
   GP1:
	UF : 1, UT : 3,		CONFIG : 'N U T, 0, 0, 0',
	X =  115.000  mm,	Y =  13.000  mm,	Z =   15.000 mm,
	W =-180.000 deg,	P =   0.000 deg,	R =    90.000 deg
};
P[1186]{
   GP1:
	UF : 1, UT : 3,		CONFIG : 'N U T, 0, 0, 0',
	X =  139.000  mm,	Y =  13.000  mm,	Z =   15.000 mm,
	W =-180.000 deg,	P =   0.000 deg,	R =    90.000 deg
};
P[1187]{
   GP1:
	UF : 1, UT : 3,		CONFIG : 'N U T, 0, 0, 0',
	X =  139.000  mm,	Y =  13.000  mm,	Z =   -1.000 mm,
	W =-180.000 deg,	P =   0.000 deg,	R =    90.000 deg
};
P[1188]{
   GP1:
	UF : 1, UT : 3,		CONFIG : 'N U T, 0, 0, 0',
	X =  139.000  mm,	Y =  13.000  mm,	Z =   15.000 mm,
	W =-180.000 deg,	P =   0.000 deg,	R =    90.000 deg
};
P[1189]{
   GP1:
	UF : 1, UT : 3,		CONFIG : 'N U T, 0, 0, 0',
	X =  142.000  mm,	Y =  13.000  mm,	Z =   15.000 mm,
	W =-180.000 deg,	P =   0.000 deg,	R =    90.000 deg
};
P[1190]{
   GP1:
	UF : 1, UT : 3,		CONFIG : 'N U T, 0, 0, 0',
	X =  142.000  mm,	Y =  13.000  mm,	Z =   -1.000 mm,
	W =-180.000 deg,	P =   0.000 deg,	R =    90.000 deg
};
P[1191]{
   GP1:
	UF : 1, UT : 3,		CONFIG : 'N U T, 0, 0, 0',
	X =  142.000  mm,	Y =  13.000  mm,	Z =   15.000 mm,
	W =-180.000 deg,	P =   0.000 deg,	R =    90.000 deg
};
P[1333]{
   GP1:
	UF : 1, UT : 3,		CONFIG : 'N U T, 0, 0, 0',
	X =  130.000  mm,	Y =  16.000  mm,	Z =   15.000 mm,
	W =-180.000 deg,	P =   0.000 deg,	R =    90.000 deg
};
P[1334]{
   GP1:
	UF : 1, UT : 3,		CONFIG : 'N U T, 0, 0, 0',
	X =  130.000  mm,	Y =  16.000  mm,	Z =   -1.000 mm,
	W =-180.000 deg,	P =   0.000 deg,	R =    90.000 deg
};
P[1335]{
   GP1:
	UF : 1, UT : 3,		CONFIG : 'N U T, 0, 0, 0',
	X =  130.000  mm,	Y =  16.000  mm,	Z =   15.000 mm,
	W =-180.000 deg,	P =   0.000 deg,	R =    90.000 deg
};
P[1336]{
   GP1:
	UF : 1, UT : 3,		CONFIG : 'N U T, 0, 0, 0',
	X =  133.000  mm,	Y =  16.000  mm,	Z =   15.000 mm,
	W =-180.000 deg,	P =   0.000 deg,	R =    90.000 deg
};
P[1337]{
   GP1:
	UF : 1, UT : 3,		CONFIG : 'N U T, 0, 0, 0',
	X =  133.000  mm,	Y =  16.000  mm,	Z =   -1.000 mm,
	W =-180.000 deg,	P =   0.000 deg,	R =    90.000 deg
};
P[1338]{
   GP1:
	UF : 1, UT : 3,		CONFIG : 'N U T, 0, 0, 0',
	X =  133.000  mm,	Y =  16.000  mm,	Z =   15.000 mm,
	W =-180.000 deg,	P =   0.000 deg,	R =    90.000 deg
};
P[1339]{
   GP1:
	UF : 1, UT : 3,		CONFIG : 'N U T, 0, 0, 0',
	X =  136.000  mm,	Y =  16.000  mm,	Z =   15.000 mm,
	W =-180.000 deg,	P =   0.000 deg,	R =    90.000 deg
};
P[1340]{
   GP1:
	UF : 1, UT : 3,		CONFIG : 'N U T, 0, 0, 0',
	X =  136.000  mm,	Y =  16.000  mm,	Z =   -1.000 mm,
	W =-180.000 deg,	P =   0.000 deg,	R =    90.000 deg
};
P[1341]{
   GP1:
	UF : 1, UT : 3,		CONFIG : 'N U T, 0, 0, 0',
	X =  136.000  mm,	Y =  16.000  mm,	Z =   15.000 mm,
	W =-180.000 deg,	P =   0.000 deg,	R =    90.000 deg
};
P[1345]{
   GP1:
	UF : 1, UT : 3,		CONFIG : 'N U T, 0, 0, 0',
	X =  142.000  mm,	Y =  16.000  mm,	Z =   15.000 mm,
	W =-180.000 deg,	P =   0.000 deg,	R =    90.000 deg
};
P[1346]{
   GP1:
	UF : 1, UT : 3,		CONFIG : 'N U T, 0, 0, 0',
	X =  142.000  mm,	Y =  16.000  mm,	Z =   -1.000 mm,
	W =-180.000 deg,	P =   0.000 deg,	R =    90.000 deg
};
P[1347]{
   GP1:
	UF : 1, UT : 3,		CONFIG : 'N U T, 0, 0, 0',
	X =  142.000  mm,	Y =  16.000  mm,	Z =   15.000 mm,
	W =-180.000 deg,	P =   0.000 deg,	R =    90.000 deg
};
P[1477]{
   GP1:
	UF : 1, UT : 3,		CONFIG : 'N U T, 0, 0, 0',
	X =  118.000  mm,	Y =  19.000  mm,	Z =   15.000 mm,
	W =-180.000 deg,	P =   0.000 deg,	R =    90.000 deg
};
P[1478]{
   GP1:
	UF : 1, UT : 3,		CONFIG : 'N U T, 0, 0, 0',
	X =  118.000  mm,	Y =  19.000  mm,	Z =   -1.000 mm,
	W =-180.000 deg,	P =   0.000 deg,	R =    90.000 deg
};
P[1479]{
   GP1:
	UF : 1, UT : 3,		CONFIG : 'N U T, 0, 0, 0',
	X =  118.000  mm,	Y =  19.000  mm,	Z =   15.000 mm,
	W =-180.000 deg,	P =   0.000 deg,	R =    90.000 deg
};
P[1480]{
   GP1:
	UF : 1, UT : 3,		CONFIG : 'N U T, 0, 0, 0',
	X =  121.000  mm,	Y =  19.000  mm,	Z =   15.000 mm,
	W =-180.000 deg,	P =   0.000 deg,	R =    90.000 deg
};
P[1481]{
   GP1:
	UF : 1, UT : 3,		CONFIG : 'N U T, 0, 0, 0',
	X =  121.000  mm,	Y =  19.000  mm,	Z =   -1.000 mm,
	W =-180.000 deg,	P =   0.000 deg,	R =    90.000 deg
};
P[1482]{
   GP1:
	UF : 1, UT : 3,		CONFIG : 'N U T, 0, 0, 0',
	X =  121.000  mm,	Y =  19.000  mm,	Z =   15.000 mm,
	W =-180.000 deg,	P =   0.000 deg,	R =    90.000 deg
};
P[1489]{
   GP1:
	UF : 1, UT : 3,		CONFIG : 'N U T, 0, 0, 0',
	X =  130.000  mm,	Y =  19.000  mm,	Z =   15.000 mm,
	W =-180.000 deg,	P =   0.000 deg,	R =    90.000 deg
};
P[1490]{
   GP1:
	UF : 1, UT : 3,		CONFIG : 'N U T, 0, 0, 0',
	X =  130.000  mm,	Y =  19.000  mm,	Z =   -1.000 mm,
	W =-180.000 deg,	P =   0.000 deg,	R =    90.000 deg
};
P[1491]{
   GP1:
	UF : 1, UT : 3,		CONFIG : 'N U T, 0, 0, 0',
	X =  130.000  mm,	Y =  19.000  mm,	Z =   15.000 mm,
	W =-180.000 deg,	P =   0.000 deg,	R =    90.000 deg
};
P[1492]{
   GP1:
	UF : 1, UT : 3,		CONFIG : 'N U T, 0, 0, 0',
	X =  133.000  mm,	Y =  19.000  mm,	Z =   15.000 mm,
	W =-180.000 deg,	P =   0.000 deg,	R =    90.000 deg
};
P[1493]{
   GP1:
	UF : 1, UT : 3,		CONFIG : 'N U T, 0, 0, 0',
	X =  133.000  mm,	Y =  19.000  mm,	Z =   -1.000 mm,
	W =-180.000 deg,	P =   0.000 deg,	R =    90.000 deg
};
P[1494]{
   GP1:
	UF : 1, UT : 3,		CONFIG : 'N U T, 0, 0, 0',
	X =  133.000  mm,	Y =  19.000  mm,	Z =   15.000 mm,
	W =-180.000 deg,	P =   0.000 deg,	R =    90.000 deg
};
P[1507]{
   GP1:
	UF : 1, UT : 3,		CONFIG : 'N U T, 0, 0, 0',
	X =  175.000  mm,	Y =  19.000  mm,	Z =   15.000 mm,
	W =-180.000 deg,	P =   0.000 deg,	R =    90.000 deg
};
P[1508]{
   GP1:
	UF : 1, UT : 3,		CONFIG : 'N U T, 0, 0, 0',
	X =  175.000  mm,	Y =  19.000  mm,	Z =   -1.000 mm,
	W =-180.000 deg,	P =   0.000 deg,	R =    90.000 deg
};
P[1509]{
   GP1:
	UF : 1, UT : 3,		CONFIG : 'N U T, 0, 0, 0',
	X =  175.000  mm,	Y =  19.000  mm,	Z =   15.000 mm,
	W =-180.000 deg,	P =   0.000 deg,	R =    90.000 deg
};
P[1627]{
   GP1:
	UF : 1, UT : 3,		CONFIG : 'N U T, 0, 0, 0',
	X =  118.000  mm,	Y =  22.000  mm,	Z =   15.000 mm,
	W =-180.000 deg,	P =   0.000 deg,	R =    90.000 deg
};
P[1628]{
   GP1:
	UF : 1, UT : 3,		CONFIG : 'N U T, 0, 0, 0',
	X =  118.000  mm,	Y =  22.000  mm,	Z =   -1.000 mm,
	W =-180.000 deg,	P =   0.000 deg,	R =    90.000 deg
};
P[1629]{
   GP1:
	UF : 1, UT : 3,		CONFIG : 'N U T, 0, 0, 0',
	X =  118.000  mm,	Y =  22.000  mm,	Z =   15.000 mm,
	W =-180.000 deg,	P =   0.000 deg,	R =    90.000 deg
};
P[1633]{
   GP1:
	UF : 1, UT : 3,		CONFIG : 'N U T, 0, 0, 0',
	X =  124.000  mm,	Y =  22.000  mm,	Z =   15.000 mm,
	W =-180.000 deg,	P =   0.000 deg,	R =    90.000 deg
};
P[1634]{
   GP1:
	UF : 1, UT : 3,		CONFIG : 'N U T, 0, 0, 0',
	X =  124.000  mm,	Y =  22.000  mm,	Z =   -1.000 mm,
	W =-180.000 deg,	P =   0.000 deg,	R =    90.000 deg
};
P[1635]{
   GP1:
	UF : 1, UT : 3,		CONFIG : 'N U T, 0, 0, 0',
	X =  124.000  mm,	Y =  22.000  mm,	Z =   15.000 mm,
	W =-180.000 deg,	P =   0.000 deg,	R =    90.000 deg
};
P[1654]{
   GP1:
	UF : 1, UT : 3,		CONFIG : 'N U T, 0, 0, 0',
	X =  175.000  mm,	Y =  22.000  mm,	Z =   15.000 mm,
	W =-180.000 deg,	P =   0.000 deg,	R =    90.000 deg
};
P[1655]{
   GP1:
	UF : 1, UT : 3,		CONFIG : 'N U T, 0, 0, 0',
	X =  175.000  mm,	Y =  22.000  mm,	Z =   -1.000 mm,
	W =-180.000 deg,	P =   0.000 deg,	R =    90.000 deg
};
P[1656]{
   GP1:
	UF : 1, UT : 3,		CONFIG : 'N U T, 0, 0, 0',
	X =  175.000  mm,	Y =  22.000  mm,	Z =   15.000 mm,
	W =-180.000 deg,	P =   0.000 deg,	R =    90.000 deg
};
P[1789]{
   GP1:
	UF : 1, UT : 3,		CONFIG : 'N U T, 0, 0, 0',
	X =  133.000  mm,	Y =  25.000  mm,	Z =   15.000 mm,
	W =-180.000 deg,	P =   0.000 deg,	R =    90.000 deg
};
P[1790]{
   GP1:
	UF : 1, UT : 3,		CONFIG : 'N U T, 0, 0, 0',
	X =  133.000  mm,	Y =  25.000  mm,	Z =   -1.000 mm,
	W =-180.000 deg,	P =   0.000 deg,	R =    90.000 deg
};
P[1791]{
   GP1:
	UF : 1, UT : 3,		CONFIG : 'N U T, 0, 0, 0',
	X =  133.000  mm,	Y =  25.000  mm,	Z =   15.000 mm,
	W =-180.000 deg,	P =   0.000 deg,	R =    90.000 deg
};
P[1798]{
   GP1:
	UF : 1, UT : 3,		CONFIG : 'N U T, 0, 0, 0',
	X =  175.000  mm,	Y =  25.000  mm,	Z =   15.000 mm,
	W =-180.000 deg,	P =   0.000 deg,	R =    90.000 deg
};
P[1799]{
   GP1:
	UF : 1, UT : 3,		CONFIG : 'N U T, 0, 0, 0',
	X =  175.000  mm,	Y =  25.000  mm,	Z =   -1.000 mm,
	W =-180.000 deg,	P =   0.000 deg,	R =    90.000 deg
};
P[1800]{
   GP1:
	UF : 1, UT : 3,		CONFIG : 'N U T, 0, 0, 0',
	X =  175.000  mm,	Y =  25.000  mm,	Z =   15.000 mm,
	W =-180.000 deg,	P =   0.000 deg,	R =    90.000 deg
};
P[1918]{
   GP1:
	UF : 1, UT : 3,		CONFIG : 'N U T, 0, 0, 0',
	X =  118.000  mm,	Y =  28.000  mm,	Z =   15.000 mm,
	W =-180.000 deg,	P =   0.000 deg,	R =    90.000 deg
};
P[1919]{
   GP1:
	UF : 1, UT : 3,		CONFIG : 'N U T, 0, 0, 0',
	X =  118.000  mm,	Y =  28.000  mm,	Z =   -1.000 mm,
	W =-180.000 deg,	P =   0.000 deg,	R =    90.000 deg
};
P[1920]{
   GP1:
	UF : 1, UT : 3,		CONFIG : 'N U T, 0, 0, 0',
	X =  118.000  mm,	Y =  28.000  mm,	Z =   15.000 mm,
	W =-180.000 deg,	P =   0.000 deg,	R =    90.000 deg
};
P[1927]{
   GP1:
	UF : 1, UT : 3,		CONFIG : 'N U T, 0, 0, 0',
	X =  127.000  mm,	Y =  28.000  mm,	Z =   15.000 mm,
	W =-180.000 deg,	P =   0.000 deg,	R =    90.000 deg
};
P[1928]{
   GP1:
	UF : 1, UT : 3,		CONFIG : 'N U T, 0, 0, 0',
	X =  127.000  mm,	Y =  28.000  mm,	Z =   -1.000 mm,
	W =-180.000 deg,	P =   0.000 deg,	R =    90.000 deg
};
P[1929]{
   GP1:
	UF : 1, UT : 3,		CONFIG : 'N U T, 0, 0, 0',
	X =  127.000  mm,	Y =  28.000  mm,	Z =   15.000 mm,
	W =-180.000 deg,	P =   0.000 deg,	R =    90.000 deg
};
P[1930]{
   GP1:
	UF : 1, UT : 3,		CONFIG : 'N U T, 0, 0, 0',
	X =  130.000  mm,	Y =  28.000  mm,	Z =   15.000 mm,
	W =-180.000 deg,	P =   0.000 deg,	R =    90.000 deg
};
P[1931]{
   GP1:
	UF : 1, UT : 3,		CONFIG : 'N U T, 0, 0, 0',
	X =  130.000  mm,	Y =  28.000  mm,	Z =   -1.000 mm,
	W =-180.000 deg,	P =   0.000 deg,	R =    90.000 deg
};
P[1932]{
   GP1:
	UF : 1, UT : 3,		CONFIG : 'N U T, 0, 0, 0',
	X =  130.000  mm,	Y =  28.000  mm,	Z =   15.000 mm,
	W =-180.000 deg,	P =   0.000 deg,	R =    90.000 deg
};
P[1939]{
   GP1:
	UF : 1, UT : 3,		CONFIG : 'N U T, 0, 0, 0',
	X =  139.000  mm,	Y =  28.000  mm,	Z =   15.000 mm,
	W =-180.000 deg,	P =   0.000 deg,	R =    90.000 deg
};
P[1940]{
   GP1:
	UF : 1, UT : 3,		CONFIG : 'N U T, 0, 0, 0',
	X =  139.000  mm,	Y =  28.000  mm,	Z =   -1.000 mm,
	W =-180.000 deg,	P =   0.000 deg,	R =    90.000 deg
};
P[1941]{
   GP1:
	UF : 1, UT : 3,		CONFIG : 'N U T, 0, 0, 0',
	X =  139.000  mm,	Y =  28.000  mm,	Z =   15.000 mm,
	W =-180.000 deg,	P =   0.000 deg,	R =    90.000 deg
};
P[2065]{
   GP1:
	UF : 1, UT : 3,		CONFIG : 'N U T, 0, 0, 0',
	X =  118.000  mm,	Y =  31.000  mm,	Z =   15.000 mm,
	W =-180.000 deg,	P =   0.000 deg,	R =    90.000 deg
};
P[2066]{
   GP1:
	UF : 1, UT : 3,		CONFIG : 'N U T, 0, 0, 0',
	X =  118.000  mm,	Y =  31.000  mm,	Z =   -1.000 mm,
	W =-180.000 deg,	P =   0.000 deg,	R =    90.000 deg
};
P[2067]{
   GP1:
	UF : 1, UT : 3,		CONFIG : 'N U T, 0, 0, 0',
	X =  118.000  mm,	Y =  31.000  mm,	Z =   15.000 mm,
	W =-180.000 deg,	P =   0.000 deg,	R =    90.000 deg
};
P[2095]{
   GP1:
	UF : 1, UT : 3,		CONFIG : 'N U T, 0, 0, 0',
	X =  175.000  mm,	Y =  31.000  mm,	Z =   15.000 mm,
	W =-180.000 deg,	P =   0.000 deg,	R =    90.000 deg
};
P[2096]{
   GP1:
	UF : 1, UT : 3,		CONFIG : 'N U T, 0, 0, 0',
	X =  175.000  mm,	Y =  31.000  mm,	Z =   -1.000 mm,
	W =-180.000 deg,	P =   0.000 deg,	R =    90.000 deg
};
P[2097]{
   GP1:
	UF : 1, UT : 3,		CONFIG : 'N U T, 0, 0, 0',
	X =  175.000  mm,	Y =  31.000  mm,	Z =   15.000 mm,
	W =-180.000 deg,	P =   0.000 deg,	R =    90.000 deg
};
P[2371]{
   GP1:
	UF : 1, UT : 3,		CONFIG : 'N U T, 0, 0, 0',
	X =  124.000  mm,	Y =  37.000  mm,	Z =   15.000 mm,
	W =-180.000 deg,	P =   0.000 deg,	R =    90.000 deg
};
P[2372]{
   GP1:
	UF : 1, UT : 3,		CONFIG : 'N U T, 0, 0, 0',
	X =  124.000  mm,	Y =  37.000  mm,	Z =   -1.000 mm,
	W =-180.000 deg,	P =   0.000 deg,	R =    90.000 deg
};
P[2373]{
   GP1:
	UF : 1, UT : 3,		CONFIG : 'N U T, 0, 0, 0',
	X =  124.000  mm,	Y =  37.000  mm,	Z =   15.000 mm,
	W =-180.000 deg,	P =   0.000 deg,	R =    90.000 deg
};
P[2374]{
   GP1:
	UF : 1, UT : 3,		CONFIG : 'N U T, 0, 0, 0',
	X =  127.000  mm,	Y =  37.000  mm,	Z =   15.000 mm,
	W =-180.000 deg,	P =   0.000 deg,	R =    90.000 deg
};
P[2375]{
   GP1:
	UF : 1, UT : 3,		CONFIG : 'N U T, 0, 0, 0',
	X =  127.000  mm,	Y =  37.000  mm,	Z =   -1.000 mm,
	W =-180.000 deg,	P =   0.000 deg,	R =    90.000 deg
};
P[2376]{
   GP1:
	UF : 1, UT : 3,		CONFIG : 'N U T, 0, 0, 0',
	X =  127.000  mm,	Y =  37.000  mm,	Z =   15.000 mm,
	W =-180.000 deg,	P =   0.000 deg,	R =    90.000 deg
};
P[2512]{
   GP1:
	UF : 1, UT : 3,		CONFIG : 'N U T, 0, 0, 0',
	X =  124.000  mm,	Y =  40.000  mm,	Z =   15.000 mm,
	W =-180.000 deg,	P =   0.000 deg,	R =    90.000 deg
};
P[2513]{
   GP1:
	UF : 1, UT : 3,		CONFIG : 'N U T, 0, 0, 0',
	X =  124.000  mm,	Y =  40.000  mm,	Z =   -1.000 mm,
	W =-180.000 deg,	P =   0.000 deg,	R =    90.000 deg
};
P[2514]{
   GP1:
	UF : 1, UT : 3,		CONFIG : 'N U T, 0, 0, 0',
	X =  124.000  mm,	Y =  40.000  mm,	Z =   15.000 mm,
	W =-180.000 deg,	P =   0.000 deg,	R =    90.000 deg
};
P[2656]{
   GP1:
	UF : 1, UT : 3,		CONFIG : 'N U T, 0, 0, 0',
	X =  130.000  mm,	Y =  43.000  mm,	Z =   15.000 mm,
	W =-180.000 deg,	P =   0.000 deg,	R =    90.000 deg
};
P[2657]{
   GP1:
	UF : 1, UT : 3,		CONFIG : 'N U T, 0, 0, 0',
	X =  130.000  mm,	Y =  43.000  mm,	Z =   -1.000 mm,
	W =-180.000 deg,	P =   0.000 deg,	R =    90.000 deg
};
P[2658]{
   GP1:
	UF : 1, UT : 3,		CONFIG : 'N U T, 0, 0, 0',
	X =  130.000  mm,	Y =  43.000  mm,	Z =   15.000 mm,
	W =-180.000 deg,	P =   0.000 deg,	R =    90.000 deg
};
P[2665]{
   GP1:
	UF : 1, UT : 3,		CONFIG : 'N U T, 0, 0, 0',
	X =  139.000  mm,	Y =  43.000  mm,	Z =   15.000 mm,
	W =-180.000 deg,	P =   0.000 deg,	R =    90.000 deg
};
P[2666]{
   GP1:
	UF : 1, UT : 3,		CONFIG : 'N U T, 0, 0, 0',
	X =  139.000  mm,	Y =  43.000  mm,	Z =   -1.000 mm,
	W =-180.000 deg,	P =   0.000 deg,	R =    90.000 deg
};
P[2667]{
   GP1:
	UF : 1, UT : 3,		CONFIG : 'N U T, 0, 0, 0',
	X =  139.000  mm,	Y =  43.000  mm,	Z =   15.000 mm,
	W =-180.000 deg,	P =   0.000 deg,	R =    90.000 deg
};
P[2803]{
   GP1:
	UF : 1, UT : 3,		CONFIG : 'N U T, 0, 0, 0',
	X =  136.000  mm,	Y =  46.000  mm,	Z =   15.000 mm,
	W =-180.000 deg,	P =   0.000 deg,	R =    90.000 deg
};
P[2804]{
   GP1:
	UF : 1, UT : 3,		CONFIG : 'N U T, 0, 0, 0',
	X =  136.000  mm,	Y =  46.000  mm,	Z =   -1.000 mm,
	W =-180.000 deg,	P =   0.000 deg,	R =    90.000 deg
};
P[2805]{
   GP1:
	UF : 1, UT : 3,		CONFIG : 'N U T, 0, 0, 0',
	X =  136.000  mm,	Y =  46.000  mm,	Z =   15.000 mm,
	W =-180.000 deg,	P =   0.000 deg,	R =    90.000 deg
};
P[3121]{
   GP1:
	UF : 1, UT : 3,		CONFIG : 'N U T, 0, 0, 0',
	X =  142.000  mm,	Y =  52.000  mm,	Z =   15.000 mm,
	W =-180.000 deg,	P =   0.000 deg,	R =    90.000 deg
};
P[3122]{
   GP1:
	UF : 1, UT : 3,		CONFIG : 'N U T, 0, 0, 0',
	X =  142.000  mm,	Y =  52.000  mm,	Z =   -1.000 mm,
	W =-180.000 deg,	P =   0.000 deg,	R =    90.000 deg
};
P[3123]{
   GP1:
	UF : 1, UT : 3,		CONFIG : 'N U T, 0, 0, 0',
	X =  142.000  mm,	Y =  52.000  mm,	Z =   15.000 mm,
	W =-180.000 deg,	P =   0.000 deg,	R =    90.000 deg
};
P[3256]{
   GP1:
	UF : 1, UT : 3,		CONFIG : 'N U T, 0, 0, 0',
	X =  127.000  mm,	Y =  55.000  mm,	Z =   15.000 mm,
	W =-180.000 deg,	P =   0.000 deg,	R =    90.000 deg
};
P[3257]{
   GP1:
	UF : 1, UT : 3,		CONFIG : 'N U T, 0, 0, 0',
	X =  127.000  mm,	Y =  55.000  mm,	Z =   -1.000 mm,
	W =-180.000 deg,	P =   0.000 deg,	R =    90.000 deg
};
P[3258]{
   GP1:
	UF : 1, UT : 3,		CONFIG : 'N U T, 0, 0, 0',
	X =  127.000  mm,	Y =  55.000  mm,	Z =   15.000 mm,
	W =-180.000 deg,	P =   0.000 deg,	R =    90.000 deg
};
P[3394]{
   GP1:
	UF : 1, UT : 3,		CONFIG : 'N U T, 0, 0, 0',
	X =  115.000  mm,	Y =  58.000  mm,	Z =   15.000 mm,
	W =-180.000 deg,	P =   0.000 deg,	R =    90.000 deg
};
P[3395]{
   GP1:
	UF : 1, UT : 3,		CONFIG : 'N U T, 0, 0, 0',
	X =  115.000  mm,	Y =  58.000  mm,	Z =   -1.000 mm,
	W =-180.000 deg,	P =   0.000 deg,	R =    90.000 deg
};
P[3396]{
   GP1:
	UF : 1, UT : 3,		CONFIG : 'N U T, 0, 0, 0',
	X =  115.000  mm,	Y =  58.000  mm,	Z =   15.000 mm,
	W =-180.000 deg,	P =   0.000 deg,	R =    90.000 deg
};
P[3397]{
   GP1:
	UF : 1, UT : 3,		CONFIG : 'N U T, 0, 0, 0',
	X =  118.000  mm,	Y =  58.000  mm,	Z =   15.000 mm,
	W =-180.000 deg,	P =   0.000 deg,	R =    90.000 deg
};
P[3398]{
   GP1:
	UF : 1, UT : 3,		CONFIG : 'N U T, 0, 0, 0',
	X =  118.000  mm,	Y =  58.000  mm,	Z =   -1.000 mm,
	W =-180.000 deg,	P =   0.000 deg,	R =    90.000 deg
};
P[3399]{
   GP1:
	UF : 1, UT : 3,		CONFIG : 'N U T, 0, 0, 0',
	X =  118.000  mm,	Y =  58.000  mm,	Z =   15.000 mm,
	W =-180.000 deg,	P =   0.000 deg,	R =    90.000 deg
};
P[3412]{
   GP1:
	UF : 1, UT : 3,		CONFIG : 'N U T, 0, 0, 0',
	X =  145.000  mm,	Y =  58.000  mm,	Z =   15.000 mm,
	W =-180.000 deg,	P =   0.000 deg,	R =    90.000 deg
};
P[3413]{
   GP1:
	UF : 1, UT : 3,		CONFIG : 'N U T, 0, 0, 0',
	X =  145.000  mm,	Y =  58.000  mm,	Z =   -1.000 mm,
	W =-180.000 deg,	P =   0.000 deg,	R =    90.000 deg
};
P[3414]{
   GP1:
	UF : 1, UT : 3,		CONFIG : 'N U T, 0, 0, 0',
	X =  145.000  mm,	Y =  58.000  mm,	Z =   15.000 mm,
	W =-180.000 deg,	P =   0.000 deg,	R =    90.000 deg
};
P[3562]{
   GP1:
	UF : 1, UT : 3,		CONFIG : 'N U T, 0, 0, 0',
	X =  172.000  mm,	Y =  61.000  mm,	Z =   15.000 mm,
	W =-180.000 deg,	P =   0.000 deg,	R =    90.000 deg
};
P[3563]{
   GP1:
	UF : 1, UT : 3,		CONFIG : 'N U T, 0, 0, 0',
	X =  172.000  mm,	Y =  61.000  mm,	Z =   -1.000 mm,
	W =-180.000 deg,	P =   0.000 deg,	R =    90.000 deg
};
P[3564]{
   GP1:
	UF : 1, UT : 3,		CONFIG : 'N U T, 0, 0, 0',
	X =  172.000  mm,	Y =  61.000  mm,	Z =   15.000 mm,
	W =-180.000 deg,	P =   0.000 deg,	R =    90.000 deg
};
P[3697]{
   GP1:
	UF : 1, UT : 3,		CONFIG : 'N U T, 0, 0, 0',
	X =  136.000  mm,	Y =  64.000  mm,	Z =   15.000 mm,
	W =-180.000 deg,	P =   0.000 deg,	R =    90.000 deg
};
P[3698]{
   GP1:
	UF : 1, UT : 3,		CONFIG : 'N U T, 0, 0, 0',
	X =  136.000  mm,	Y =  64.000  mm,	Z =   -1.000 mm,
	W =-180.000 deg,	P =   0.000 deg,	R =    90.000 deg
};
P[3699]{
   GP1:
	UF : 1, UT : 3,		CONFIG : 'N U T, 0, 0, 0',
	X =  136.000  mm,	Y =  64.000  mm,	Z =   15.000 mm,
	W =-180.000 deg,	P =   0.000 deg,	R =    90.000 deg
};
P[3832]{
   GP1:
	UF : 1, UT : 3,		CONFIG : 'N U T, 0, 0, 0',
	X =  133.000  mm,	Y =  67.000  mm,	Z =   15.000 mm,
	W =-180.000 deg,	P =   0.000 deg,	R =    90.000 deg
};
P[3833]{
   GP1:
	UF : 1, UT : 3,		CONFIG : 'N U T, 0, 0, 0',
	X =  133.000  mm,	Y =  67.000  mm,	Z =   -1.000 mm,
	W =-180.000 deg,	P =   0.000 deg,	R =    90.000 deg
};
P[3834]{
   GP1:
	UF : 1, UT : 3,		CONFIG : 'N U T, 0, 0, 0',
	X =  133.000  mm,	Y =  67.000  mm,	Z =   15.000 mm,
	W =-180.000 deg,	P =   0.000 deg,	R =    90.000 deg
};
P[3979]{
   GP1:
	UF : 1, UT : 3,		CONFIG : 'N U T, 0, 0, 0',
	X =  142.000  mm,	Y =  70.000  mm,	Z =   15.000 mm,
	W =-180.000 deg,	P =   0.000 deg,	R =    90.000 deg
};
P[3980]{
   GP1:
	UF : 1, UT : 3,		CONFIG : 'N U T, 0, 0, 0',
	X =  142.000  mm,	Y =  70.000  mm,	Z =   -1.000 mm,
	W =-180.000 deg,	P =   0.000 deg,	R =    90.000 deg
};
P[3981]{
   GP1:
	UF : 1, UT : 3,		CONFIG : 'N U T, 0, 0, 0',
	X =  142.000  mm,	Y =  70.000  mm,	Z =   15.000 mm,
	W =-180.000 deg,	P =   0.000 deg,	R =    90.000 deg
};
P[4114]{
   GP1:
	UF : 1, UT : 3,		CONFIG : 'N U T, 0, 0, 0',
	X =  142.000  mm,	Y =  73.000  mm,	Z =   15.000 mm,
	W =-180.000 deg,	P =   0.000 deg,	R =    90.000 deg
};
P[4115]{
   GP1:
	UF : 1, UT : 3,		CONFIG : 'N U T, 0, 0, 0',
	X =  142.000  mm,	Y =  73.000  mm,	Z =   -1.000 mm,
	W =-180.000 deg,	P =   0.000 deg,	R =    90.000 deg
};
P[4116]{
   GP1:
	UF : 1, UT : 3,		CONFIG : 'N U T, 0, 0, 0',
	X =  142.000  mm,	Y =  73.000  mm,	Z =   15.000 mm,
	W =-180.000 deg,	P =   0.000 deg,	R =    90.000 deg
};
P[4123]{
   GP1:
	UF : 1, UT : 3,		CONFIG : 'N U T, 0, 0, 0',
	X =  169.000  mm,	Y =  73.000  mm,	Z =   15.000 mm,
	W =-180.000 deg,	P =   0.000 deg,	R =    90.000 deg
};
P[4124]{
   GP1:
	UF : 1, UT : 3,		CONFIG : 'N U T, 0, 0, 0',
	X =  169.000  mm,	Y =  73.000  mm,	Z =   -1.000 mm,
	W =-180.000 deg,	P =   0.000 deg,	R =    90.000 deg
};
P[4125]{
   GP1:
	UF : 1, UT : 3,		CONFIG : 'N U T, 0, 0, 0',
	X =  169.000  mm,	Y =  73.000  mm,	Z =   15.000 mm,
	W =-180.000 deg,	P =   0.000 deg,	R =    90.000 deg
};
P[4288]{
   GP1:
	UF : 1, UT : 3,		CONFIG : 'N U T, 0, 0, 0',
	X =  31.000  mm,	Y =  79.000  mm,	Z =   15.000 mm,
	W =-180.000 deg,	P =   0.000 deg,	R =    90.000 deg
};
P[4289]{
   GP1:
	UF : 1, UT : 3,		CONFIG : 'N U T, 0, 0, 0',
	X =  31.000  mm,	Y =  79.000  mm,	Z =   -1.000 mm,
	W =-180.000 deg,	P =   0.000 deg,	R =    90.000 deg
};
P[4290]{
   GP1:
	UF : 1, UT : 3,		CONFIG : 'N U T, 0, 0, 0',
	X =  31.000  mm,	Y =  79.000  mm,	Z =   15.000 mm,
	W =-180.000 deg,	P =   0.000 deg,	R =    90.000 deg
};
P[4366]{
   GP1:
	UF : 1, UT : 3,		CONFIG : 'N U T, 0, 0, 0',
	X =  118.000  mm,	Y =  79.000  mm,	Z =   15.000 mm,
	W =-180.000 deg,	P =   0.000 deg,	R =    90.000 deg
};
P[4367]{
   GP1:
	UF : 1, UT : 3,		CONFIG : 'N U T, 0, 0, 0',
	X =  118.000  mm,	Y =  79.000  mm,	Z =   -1.000 mm,
	W =-180.000 deg,	P =   0.000 deg,	R =    90.000 deg
};
P[4368]{
   GP1:
	UF : 1, UT : 3,		CONFIG : 'N U T, 0, 0, 0',
	X =  118.000  mm,	Y =  79.000  mm,	Z =   15.000 mm,
	W =-180.000 deg,	P =   0.000 deg,	R =    90.000 deg
};
P[4384]{
   GP1:
	UF : 1, UT : 3,		CONFIG : 'N U T, 0, 0, 0',
	X =  145.000  mm,	Y =  79.000  mm,	Z =   15.000 mm,
	W =-180.000 deg,	P =   0.000 deg,	R =    90.000 deg
};
P[4385]{
   GP1:
	UF : 1, UT : 3,		CONFIG : 'N U T, 0, 0, 0',
	X =  145.000  mm,	Y =  79.000  mm,	Z =   -1.000 mm,
	W =-180.000 deg,	P =   0.000 deg,	R =    90.000 deg
};
P[4386]{
   GP1:
	UF : 1, UT : 3,		CONFIG : 'N U T, 0, 0, 0',
	X =  145.000  mm,	Y =  79.000  mm,	Z =   15.000 mm,
	W =-180.000 deg,	P =   0.000 deg,	R =    90.000 deg
};
P[4432]{
   GP1:
	UF : 1, UT : 3,		CONFIG : 'N U T, 0, 0, 0',
	X =  37.000  mm,	Y =  82.000  mm,	Z =   15.000 mm,
	W =-180.000 deg,	P =   0.000 deg,	R =    90.000 deg
};
P[4433]{
   GP1:
	UF : 1, UT : 3,		CONFIG : 'N U T, 0, 0, 0',
	X =  37.000  mm,	Y =  82.000  mm,	Z =   -1.000 mm,
	W =-180.000 deg,	P =   0.000 deg,	R =    90.000 deg
};
P[4434]{
   GP1:
	UF : 1, UT : 3,		CONFIG : 'N U T, 0, 0, 0',
	X =  37.000  mm,	Y =  82.000  mm,	Z =   15.000 mm,
	W =-180.000 deg,	P =   0.000 deg,	R =    90.000 deg
};
P[4585]{
   GP1:
	UF : 1, UT : 3,		CONFIG : 'N U T, 0, 0, 0',
	X =  43.000  mm,	Y =  85.000  mm,	Z =   15.000 mm,
	W =-180.000 deg,	P =   0.000 deg,	R =    90.000 deg
};
P[4586]{
   GP1:
	UF : 1, UT : 3,		CONFIG : 'N U T, 0, 0, 0',
	X =  43.000  mm,	Y =  85.000  mm,	Z =   -1.000 mm,
	W =-180.000 deg,	P =   0.000 deg,	R =    90.000 deg
};
P[4587]{
   GP1:
	UF : 1, UT : 3,		CONFIG : 'N U T, 0, 0, 0',
	X =  43.000  mm,	Y =  85.000  mm,	Z =   15.000 mm,
	W =-180.000 deg,	P =   0.000 deg,	R =    90.000 deg
};
P[4669]{
   GP1:
	UF : 1, UT : 3,		CONFIG : 'N U T, 0, 0, 0',
	X =  139.000  mm,	Y =  85.000  mm,	Z =   15.000 mm,
	W =-180.000 deg,	P =   0.000 deg,	R =    90.000 deg
};
P[4670]{
   GP1:
	UF : 1, UT : 3,		CONFIG : 'N U T, 0, 0, 0',
	X =  139.000  mm,	Y =  85.000  mm,	Z =   -1.000 mm,
	W =-180.000 deg,	P =   0.000 deg,	R =    90.000 deg
};
P[4671]{
   GP1:
	UF : 1, UT : 3,		CONFIG : 'N U T, 0, 0, 0',
	X =  139.000  mm,	Y =  85.000  mm,	Z =   15.000 mm,
	W =-180.000 deg,	P =   0.000 deg,	R =    90.000 deg
};
P[4675]{
   GP1:
	UF : 1, UT : 3,		CONFIG : 'N U T, 0, 0, 0',
	X =  145.000  mm,	Y =  85.000  mm,	Z =   15.000 mm,
	W =-180.000 deg,	P =   0.000 deg,	R =    90.000 deg
};
P[4676]{
   GP1:
	UF : 1, UT : 3,		CONFIG : 'N U T, 0, 0, 0',
	X =  145.000  mm,	Y =  85.000  mm,	Z =   -1.000 mm,
	W =-180.000 deg,	P =   0.000 deg,	R =    90.000 deg
};
P[4677]{
   GP1:
	UF : 1, UT : 3,		CONFIG : 'N U T, 0, 0, 0',
	X =  145.000  mm,	Y =  85.000  mm,	Z =   15.000 mm,
	W =-180.000 deg,	P =   0.000 deg,	R =    90.000 deg
};
P[4717]{
   GP1:
	UF : 1, UT : 3,		CONFIG : 'N U T, 0, 0, 0',
	X =  22.000  mm,	Y =  88.000  mm,	Z =   15.000 mm,
	W =-180.000 deg,	P =   0.000 deg,	R =    90.000 deg
};
P[4718]{
   GP1:
	UF : 1, UT : 3,		CONFIG : 'N U T, 0, 0, 0',
	X =  22.000  mm,	Y =  88.000  mm,	Z =   -1.000 mm,
	W =-180.000 deg,	P =   0.000 deg,	R =    90.000 deg
};
P[4719]{
   GP1:
	UF : 1, UT : 3,		CONFIG : 'N U T, 0, 0, 0',
	X =  22.000  mm,	Y =  88.000  mm,	Z =   15.000 mm,
	W =-180.000 deg,	P =   0.000 deg,	R =    90.000 deg
};
P[4729]{
   GP1:
	UF : 1, UT : 3,		CONFIG : 'N U T, 0, 0, 0',
	X =  34.000  mm,	Y =  88.000  mm,	Z =   15.000 mm,
	W =-180.000 deg,	P =   0.000 deg,	R =    90.000 deg
};
P[4730]{
   GP1:
	UF : 1, UT : 3,		CONFIG : 'N U T, 0, 0, 0',
	X =  34.000  mm,	Y =  88.000  mm,	Z =   -1.000 mm,
	W =-180.000 deg,	P =   0.000 deg,	R =    90.000 deg
};
P[4731]{
   GP1:
	UF : 1, UT : 3,		CONFIG : 'N U T, 0, 0, 0',
	X =  34.000  mm,	Y =  88.000  mm,	Z =   15.000 mm,
	W =-180.000 deg,	P =   0.000 deg,	R =    90.000 deg
};
P[4732]{
   GP1:
	UF : 1, UT : 3,		CONFIG : 'N U T, 0, 0, 0',
	X =  37.000  mm,	Y =  88.000  mm,	Z =   15.000 mm,
	W =-180.000 deg,	P =   0.000 deg,	R =    90.000 deg
};
P[4733]{
   GP1:
	UF : 1, UT : 3,		CONFIG : 'N U T, 0, 0, 0',
	X =  37.000  mm,	Y =  88.000  mm,	Z =   -1.000 mm,
	W =-180.000 deg,	P =   0.000 deg,	R =    90.000 deg
};
P[4734]{
   GP1:
	UF : 1, UT : 3,		CONFIG : 'N U T, 0, 0, 0',
	X =  37.000  mm,	Y =  88.000  mm,	Z =   15.000 mm,
	W =-180.000 deg,	P =   0.000 deg,	R =    90.000 deg
};
P[4735]{
   GP1:
	UF : 1, UT : 3,		CONFIG : 'N U T, 0, 0, 0',
	X =  40.000  mm,	Y =  88.000  mm,	Z =   15.000 mm,
	W =-180.000 deg,	P =   0.000 deg,	R =    90.000 deg
};
P[4736]{
   GP1:
	UF : 1, UT : 3,		CONFIG : 'N U T, 0, 0, 0',
	X =  40.000  mm,	Y =  88.000  mm,	Z =   -1.000 mm,
	W =-180.000 deg,	P =   0.000 deg,	R =    90.000 deg
};
P[4737]{
   GP1:
	UF : 1, UT : 3,		CONFIG : 'N U T, 0, 0, 0',
	X =  40.000  mm,	Y =  88.000  mm,	Z =   15.000 mm,
	W =-180.000 deg,	P =   0.000 deg,	R =    90.000 deg
};
P[4741]{
   GP1:
	UF : 1, UT : 3,		CONFIG : 'N U T, 0, 0, 0',
	X =  46.000  mm,	Y =  88.000  mm,	Z =   15.000 mm,
	W =-180.000 deg,	P =   0.000 deg,	R =    90.000 deg
};
P[4742]{
   GP1:
	UF : 1, UT : 3,		CONFIG : 'N U T, 0, 0, 0',
	X =  46.000  mm,	Y =  88.000  mm,	Z =   -1.000 mm,
	W =-180.000 deg,	P =   0.000 deg,	R =    90.000 deg
};
P[4743]{
   GP1:
	UF : 1, UT : 3,		CONFIG : 'N U T, 0, 0, 0',
	X =  46.000  mm,	Y =  88.000  mm,	Z =   15.000 mm,
	W =-180.000 deg,	P =   0.000 deg,	R =    90.000 deg
};
P[4855]{
   GP1:
	UF : 1, UT : 3,		CONFIG : 'N U T, 0, 0, 0',
	X =  16.000  mm,	Y =  91.000  mm,	Z =   15.000 mm,
	W =-180.000 deg,	P =   0.000 deg,	R =    90.000 deg
};
P[4856]{
   GP1:
	UF : 1, UT : 3,		CONFIG : 'N U T, 0, 0, 0',
	X =  16.000  mm,	Y =  91.000  mm,	Z =   -1.000 mm,
	W =-180.000 deg,	P =   0.000 deg,	R =    90.000 deg
};
P[4857]{
   GP1:
	UF : 1, UT : 3,		CONFIG : 'N U T, 0, 0, 0',
	X =  16.000  mm,	Y =  91.000  mm,	Z =   15.000 mm,
	W =-180.000 deg,	P =   0.000 deg,	R =    90.000 deg
};
P[4858]{
   GP1:
	UF : 1, UT : 3,		CONFIG : 'N U T, 0, 0, 0',
	X =  19.000  mm,	Y =  91.000  mm,	Z =   15.000 mm,
	W =-180.000 deg,	P =   0.000 deg,	R =    90.000 deg
};
P[4859]{
   GP1:
	UF : 1, UT : 3,		CONFIG : 'N U T, 0, 0, 0',
	X =  19.000  mm,	Y =  91.000  mm,	Z =   -1.000 mm,
	W =-180.000 deg,	P =   0.000 deg,	R =    90.000 deg
};
P[4860]{
   GP1:
	UF : 1, UT : 3,		CONFIG : 'N U T, 0, 0, 0',
	X =  19.000  mm,	Y =  91.000  mm,	Z =   15.000 mm,
	W =-180.000 deg,	P =   0.000 deg,	R =    90.000 deg
};
P[4861]{
   GP1:
	UF : 1, UT : 3,		CONFIG : 'N U T, 0, 0, 0',
	X =  22.000  mm,	Y =  91.000  mm,	Z =   15.000 mm,
	W =-180.000 deg,	P =   0.000 deg,	R =    90.000 deg
};
P[4862]{
   GP1:
	UF : 1, UT : 3,		CONFIG : 'N U T, 0, 0, 0',
	X =  22.000  mm,	Y =  91.000  mm,	Z =   -1.000 mm,
	W =-180.000 deg,	P =   0.000 deg,	R =    90.000 deg
};
P[4863]{
   GP1:
	UF : 1, UT : 3,		CONFIG : 'N U T, 0, 0, 0',
	X =  22.000  mm,	Y =  91.000  mm,	Z =   15.000 mm,
	W =-180.000 deg,	P =   0.000 deg,	R =    90.000 deg
};
P[4864]{
   GP1:
	UF : 1, UT : 3,		CONFIG : 'N U T, 0, 0, 0',
	X =  25.000  mm,	Y =  91.000  mm,	Z =   15.000 mm,
	W =-180.000 deg,	P =   0.000 deg,	R =    90.000 deg
};
P[4865]{
   GP1:
	UF : 1, UT : 3,		CONFIG : 'N U T, 0, 0, 0',
	X =  25.000  mm,	Y =  91.000  mm,	Z =   -1.000 mm,
	W =-180.000 deg,	P =   0.000 deg,	R =    90.000 deg
};
P[4866]{
   GP1:
	UF : 1, UT : 3,		CONFIG : 'N U T, 0, 0, 0',
	X =  25.000  mm,	Y =  91.000  mm,	Z =   15.000 mm,
	W =-180.000 deg,	P =   0.000 deg,	R =    90.000 deg
};
P[4870]{
   GP1:
	UF : 1, UT : 3,		CONFIG : 'N U T, 0, 0, 0',
	X =  31.000  mm,	Y =  91.000  mm,	Z =   15.000 mm,
	W =-180.000 deg,	P =   0.000 deg,	R =    90.000 deg
};
P[4871]{
   GP1:
	UF : 1, UT : 3,		CONFIG : 'N U T, 0, 0, 0',
	X =  31.000  mm,	Y =  91.000  mm,	Z =   -1.000 mm,
	W =-180.000 deg,	P =   0.000 deg,	R =    90.000 deg
};
P[4872]{
   GP1:
	UF : 1, UT : 3,		CONFIG : 'N U T, 0, 0, 0',
	X =  31.000  mm,	Y =  91.000  mm,	Z =   15.000 mm,
	W =-180.000 deg,	P =   0.000 deg,	R =    90.000 deg
};
P[4873]{
   GP1:
	UF : 1, UT : 3,		CONFIG : 'N U T, 0, 0, 0',
	X =  34.000  mm,	Y =  91.000  mm,	Z =   15.000 mm,
	W =-180.000 deg,	P =   0.000 deg,	R =    90.000 deg
};
P[4874]{
   GP1:
	UF : 1, UT : 3,		CONFIG : 'N U T, 0, 0, 0',
	X =  34.000  mm,	Y =  91.000  mm,	Z =   -1.000 mm,
	W =-180.000 deg,	P =   0.000 deg,	R =    90.000 deg
};
P[4875]{
   GP1:
	UF : 1, UT : 3,		CONFIG : 'N U T, 0, 0, 0',
	X =  34.000  mm,	Y =  91.000  mm,	Z =   15.000 mm,
	W =-180.000 deg,	P =   0.000 deg,	R =    90.000 deg
};
P[4876]{
   GP1:
	UF : 1, UT : 3,		CONFIG : 'N U T, 0, 0, 0',
	X =  37.000  mm,	Y =  91.000  mm,	Z =   15.000 mm,
	W =-180.000 deg,	P =   0.000 deg,	R =    90.000 deg
};
P[4877]{
   GP1:
	UF : 1, UT : 3,		CONFIG : 'N U T, 0, 0, 0',
	X =  37.000  mm,	Y =  91.000  mm,	Z =   -1.000 mm,
	W =-180.000 deg,	P =   0.000 deg,	R =    90.000 deg
};
P[4878]{
   GP1:
	UF : 1, UT : 3,		CONFIG : 'N U T, 0, 0, 0',
	X =  37.000  mm,	Y =  91.000  mm,	Z =   15.000 mm,
	W =-180.000 deg,	P =   0.000 deg,	R =    90.000 deg
};
P[4879]{
   GP1:
	UF : 1, UT : 3,		CONFIG : 'N U T, 0, 0, 0',
	X =  40.000  mm,	Y =  91.000  mm,	Z =   15.000 mm,
	W =-180.000 deg,	P =   0.000 deg,	R =    90.000 deg
};
P[4880]{
   GP1:
	UF : 1, UT : 3,		CONFIG : 'N U T, 0, 0, 0',
	X =  40.000  mm,	Y =  91.000  mm,	Z =   -1.000 mm,
	W =-180.000 deg,	P =   0.000 deg,	R =    90.000 deg
};
P[4881]{
   GP1:
	UF : 1, UT : 3,		CONFIG : 'N U T, 0, 0, 0',
	X =  40.000  mm,	Y =  91.000  mm,	Z =   15.000 mm,
	W =-180.000 deg,	P =   0.000 deg,	R =    90.000 deg
};
P[4882]{
   GP1:
	UF : 1, UT : 3,		CONFIG : 'N U T, 0, 0, 0',
	X =  43.000  mm,	Y =  91.000  mm,	Z =   15.000 mm,
	W =-180.000 deg,	P =   0.000 deg,	R =    90.000 deg
};
P[4883]{
   GP1:
	UF : 1, UT : 3,		CONFIG : 'N U T, 0, 0, 0',
	X =  43.000  mm,	Y =  91.000  mm,	Z =   -1.000 mm,
	W =-180.000 deg,	P =   0.000 deg,	R =    90.000 deg
};
P[4884]{
   GP1:
	UF : 1, UT : 3,		CONFIG : 'N U T, 0, 0, 0',
	X =  43.000  mm,	Y =  91.000  mm,	Z =   15.000 mm,
	W =-180.000 deg,	P =   0.000 deg,	R =    90.000 deg
};
P[4885]{
   GP1:
	UF : 1, UT : 3,		CONFIG : 'N U T, 0, 0, 0',
	X =  46.000  mm,	Y =  91.000  mm,	Z =   15.000 mm,
	W =-180.000 deg,	P =   0.000 deg,	R =    90.000 deg
};
P[4886]{
   GP1:
	UF : 1, UT : 3,		CONFIG : 'N U T, 0, 0, 0',
	X =  46.000  mm,	Y =  91.000  mm,	Z =   -1.000 mm,
	W =-180.000 deg,	P =   0.000 deg,	R =    90.000 deg
};
P[4887]{
   GP1:
	UF : 1, UT : 3,		CONFIG : 'N U T, 0, 0, 0',
	X =  46.000  mm,	Y =  91.000  mm,	Z =   15.000 mm,
	W =-180.000 deg,	P =   0.000 deg,	R =    90.000 deg
};
P[4888]{
   GP1:
	UF : 1, UT : 3,		CONFIG : 'N U T, 0, 0, 0',
	X =  49.000  mm,	Y =  91.000  mm,	Z =   15.000 mm,
	W =-180.000 deg,	P =   0.000 deg,	R =    90.000 deg
};
P[4889]{
   GP1:
	UF : 1, UT : 3,		CONFIG : 'N U T, 0, 0, 0',
	X =  49.000  mm,	Y =  91.000  mm,	Z =   -1.000 mm,
	W =-180.000 deg,	P =   0.000 deg,	R =    90.000 deg
};
P[4890]{
   GP1:
	UF : 1, UT : 3,		CONFIG : 'N U T, 0, 0, 0',
	X =  49.000  mm,	Y =  91.000  mm,	Z =   15.000 mm,
	W =-180.000 deg,	P =   0.000 deg,	R =    90.000 deg
};
P[4963]{
   GP1:
	UF : 1, UT : 3,		CONFIG : 'N U T, 0, 0, 0',
	X =  136.000  mm,	Y =  91.000  mm,	Z =   15.000 mm,
	W =-180.000 deg,	P =   0.000 deg,	R =    90.000 deg
};
P[4964]{
   GP1:
	UF : 1, UT : 3,		CONFIG : 'N U T, 0, 0, 0',
	X =  136.000  mm,	Y =  91.000  mm,	Z =   -1.000 mm,
	W =-180.000 deg,	P =   0.000 deg,	R =    90.000 deg
};
P[4965]{
   GP1:
	UF : 1, UT : 3,		CONFIG : 'N U T, 0, 0, 0',
	X =  136.000  mm,	Y =  91.000  mm,	Z =   15.000 mm,
	W =-180.000 deg,	P =   0.000 deg,	R =    90.000 deg
};
P[5002]{
   GP1:
	UF : 1, UT : 3,		CONFIG : 'N U T, 0, 0, 0',
	X =  16.000  mm,	Y =  94.000  mm,	Z =   15.000 mm,
	W =-180.000 deg,	P =   0.000 deg,	R =    90.000 deg
};
P[5003]{
   GP1:
	UF : 1, UT : 3,		CONFIG : 'N U T, 0, 0, 0',
	X =  16.000  mm,	Y =  94.000  mm,	Z =   -1.000 mm,
	W =-180.000 deg,	P =   0.000 deg,	R =    90.000 deg
};
P[5004]{
   GP1:
	UF : 1, UT : 3,		CONFIG : 'N U T, 0, 0, 0',
	X =  16.000  mm,	Y =  94.000  mm,	Z =   15.000 mm,
	W =-180.000 deg,	P =   0.000 deg,	R =    90.000 deg
};
P[5005]{
   GP1:
	UF : 1, UT : 3,		CONFIG : 'N U T, 0, 0, 0',
	X =  19.000  mm,	Y =  94.000  mm,	Z =   15.000 mm,
	W =-180.000 deg,	P =   0.000 deg,	R =    90.000 deg
};
P[5006]{
   GP1:
	UF : 1, UT : 3,		CONFIG : 'N U T, 0, 0, 0',
	X =  19.000  mm,	Y =  94.000  mm,	Z =   -1.000 mm,
	W =-180.000 deg,	P =   0.000 deg,	R =    90.000 deg
};
P[5007]{
   GP1:
	UF : 1, UT : 3,		CONFIG : 'N U T, 0, 0, 0',
	X =  19.000  mm,	Y =  94.000  mm,	Z =   15.000 mm,
	W =-180.000 deg,	P =   0.000 deg,	R =    90.000 deg
};
P[5011]{
   GP1:
	UF : 1, UT : 3,		CONFIG : 'N U T, 0, 0, 0',
	X =  25.000  mm,	Y =  94.000  mm,	Z =   15.000 mm,
	W =-180.000 deg,	P =   0.000 deg,	R =    90.000 deg
};
P[5012]{
   GP1:
	UF : 1, UT : 3,		CONFIG : 'N U T, 0, 0, 0',
	X =  25.000  mm,	Y =  94.000  mm,	Z =   -1.000 mm,
	W =-180.000 deg,	P =   0.000 deg,	R =    90.000 deg
};
P[5013]{
   GP1:
	UF : 1, UT : 3,		CONFIG : 'N U T, 0, 0, 0',
	X =  25.000  mm,	Y =  94.000  mm,	Z =   15.000 mm,
	W =-180.000 deg,	P =   0.000 deg,	R =    90.000 deg
};
P[5032]{
   GP1:
	UF : 1, UT : 3,		CONFIG : 'N U T, 0, 0, 0',
	X =  46.000  mm,	Y =  94.000  mm,	Z =   15.000 mm,
	W =-180.000 deg,	P =   0.000 deg,	R =    90.000 deg
};
P[5033]{
   GP1:
	UF : 1, UT : 3,		CONFIG : 'N U T, 0, 0, 0',
	X =  46.000  mm,	Y =  94.000  mm,	Z =   -1.000 mm,
	W =-180.000 deg,	P =   0.000 deg,	R =    90.000 deg
};
P[5034]{
   GP1:
	UF : 1, UT : 3,		CONFIG : 'N U T, 0, 0, 0',
	X =  46.000  mm,	Y =  94.000  mm,	Z =   15.000 mm,
	W =-180.000 deg,	P =   0.000 deg,	R =    90.000 deg
};
P[5095]{
   GP1:
	UF : 1, UT : 3,		CONFIG : 'N U T, 0, 0, 0',
	X =  130.000  mm,	Y =  94.000  mm,	Z =   15.000 mm,
	W =-180.000 deg,	P =   0.000 deg,	R =    90.000 deg
};
P[5096]{
   GP1:
	UF : 1, UT : 3,		CONFIG : 'N U T, 0, 0, 0',
	X =  130.000  mm,	Y =  94.000  mm,	Z =   -1.000 mm,
	W =-180.000 deg,	P =   0.000 deg,	R =    90.000 deg
};
P[5097]{
   GP1:
	UF : 1, UT : 3,		CONFIG : 'N U T, 0, 0, 0',
	X =  130.000  mm,	Y =  94.000  mm,	Z =   15.000 mm,
	W =-180.000 deg,	P =   0.000 deg,	R =    90.000 deg
};
P[5098]{
   GP1:
	UF : 1, UT : 3,		CONFIG : 'N U T, 0, 0, 0',
	X =  133.000  mm,	Y =  94.000  mm,	Z =   15.000 mm,
	W =-180.000 deg,	P =   0.000 deg,	R =    90.000 deg
};
P[5099]{
   GP1:
	UF : 1, UT : 3,		CONFIG : 'N U T, 0, 0, 0',
	X =  133.000  mm,	Y =  94.000  mm,	Z =   -1.000 mm,
	W =-180.000 deg,	P =   0.000 deg,	R =    90.000 deg
};
P[5100]{
   GP1:
	UF : 1, UT : 3,		CONFIG : 'N U T, 0, 0, 0',
	X =  133.000  mm,	Y =  94.000  mm,	Z =   15.000 mm,
	W =-180.000 deg,	P =   0.000 deg,	R =    90.000 deg
};
P[5143]{
   GP1:
	UF : 1, UT : 3,		CONFIG : 'N U T, 0, 0, 0',
	X =  16.000  mm,	Y =  97.000  mm,	Z =   15.000 mm,
	W =-180.000 deg,	P =   0.000 deg,	R =    90.000 deg
};
P[5144]{
   GP1:
	UF : 1, UT : 3,		CONFIG : 'N U T, 0, 0, 0',
	X =  16.000  mm,	Y =  97.000  mm,	Z =   -1.000 mm,
	W =-180.000 deg,	P =   0.000 deg,	R =    90.000 deg
};
P[5145]{
   GP1:
	UF : 1, UT : 3,		CONFIG : 'N U T, 0, 0, 0',
	X =  16.000  mm,	Y =  97.000  mm,	Z =   15.000 mm,
	W =-180.000 deg,	P =   0.000 deg,	R =    90.000 deg
};
P[5149]{
   GP1:
	UF : 1, UT : 3,		CONFIG : 'N U T, 0, 0, 0',
	X =  22.000  mm,	Y =  97.000  mm,	Z =   15.000 mm,
	W =-180.000 deg,	P =   0.000 deg,	R =    90.000 deg
};
P[5150]{
   GP1:
	UF : 1, UT : 3,		CONFIG : 'N U T, 0, 0, 0',
	X =  22.000  mm,	Y =  97.000  mm,	Z =   -1.000 mm,
	W =-180.000 deg,	P =   0.000 deg,	R =    90.000 deg
};
P[5151]{
   GP1:
	UF : 1, UT : 3,		CONFIG : 'N U T, 0, 0, 0',
	X =  22.000  mm,	Y =  97.000  mm,	Z =   15.000 mm,
	W =-180.000 deg,	P =   0.000 deg,	R =    90.000 deg
};
P[5152]{
   GP1:
	UF : 1, UT : 3,		CONFIG : 'N U T, 0, 0, 0',
	X =  25.000  mm,	Y =  97.000  mm,	Z =   15.000 mm,
	W =-180.000 deg,	P =   0.000 deg,	R =    90.000 deg
};
P[5153]{
   GP1:
	UF : 1, UT : 3,		CONFIG : 'N U T, 0, 0, 0',
	X =  25.000  mm,	Y =  97.000  mm,	Z =   -1.000 mm,
	W =-180.000 deg,	P =   0.000 deg,	R =    90.000 deg
};
P[5154]{
   GP1:
	UF : 1, UT : 3,		CONFIG : 'N U T, 0, 0, 0',
	X =  25.000  mm,	Y =  97.000  mm,	Z =   15.000 mm,
	W =-180.000 deg,	P =   0.000 deg,	R =    90.000 deg
};
P[5245]{
   GP1:
	UF : 1, UT : 3,		CONFIG : 'N U T, 0, 0, 0',
	X =  118.000  mm,	Y =  97.000  mm,	Z =   15.000 mm,
	W =-180.000 deg,	P =   0.000 deg,	R =    90.000 deg
};
P[5246]{
   GP1:
	UF : 1, UT : 3,		CONFIG : 'N U T, 0, 0, 0',
	X =  118.000  mm,	Y =  97.000  mm,	Z =   -1.000 mm,
	W =-180.000 deg,	P =   0.000 deg,	R =    90.000 deg
};
P[5247]{
   GP1:
	UF : 1, UT : 3,		CONFIG : 'N U T, 0, 0, 0',
	X =  118.000  mm,	Y =  97.000  mm,	Z =   15.000 mm,
	W =-180.000 deg,	P =   0.000 deg,	R =    90.000 deg
};
P[5254]{
   GP1:
	UF : 1, UT : 3,		CONFIG : 'N U T, 0, 0, 0',
	X =  127.000  mm,	Y =  97.000  mm,	Z =   15.000 mm,
	W =-180.000 deg,	P =   0.000 deg,	R =    90.000 deg
};
P[5255]{
   GP1:
	UF : 1, UT : 3,		CONFIG : 'N U T, 0, 0, 0',
	X =  127.000  mm,	Y =  97.000  mm,	Z =   -1.000 mm,
	W =-180.000 deg,	P =   0.000 deg,	R =    90.000 deg
};
P[5256]{
   GP1:
	UF : 1, UT : 3,		CONFIG : 'N U T, 0, 0, 0',
	X =  127.000  mm,	Y =  97.000  mm,	Z =   15.000 mm,
	W =-180.000 deg,	P =   0.000 deg,	R =    90.000 deg
};
P[5326]{
   GP1:
	UF : 1, UT : 3,		CONFIG : 'N U T, 0, 0, 0',
	X =  31.000  mm,	Y =  100.000  mm,	Z =   15.000 mm,
	W =-180.000 deg,	P =   0.000 deg,	R =    90.000 deg
};
P[5327]{
   GP1:
	UF : 1, UT : 3,		CONFIG : 'N U T, 0, 0, 0',
	X =  31.000  mm,	Y =  100.000  mm,	Z =   -1.000 mm,
	W =-180.000 deg,	P =   0.000 deg,	R =    90.000 deg
};
P[5328]{
   GP1:
	UF : 1, UT : 3,		CONFIG : 'N U T, 0, 0, 0',
	X =  31.000  mm,	Y =  100.000  mm,	Z =   15.000 mm,
	W =-180.000 deg,	P =   0.000 deg,	R =    90.000 deg
};
P[5329]{
   GP1:
	UF : 1, UT : 3,		CONFIG : 'N U T, 0, 0, 0',
	X =  34.000  mm,	Y =  100.000  mm,	Z =   15.000 mm,
	W =-180.000 deg,	P =   0.000 deg,	R =    90.000 deg
};
P[5330]{
   GP1:
	UF : 1, UT : 3,		CONFIG : 'N U T, 0, 0, 0',
	X =  34.000  mm,	Y =  100.000  mm,	Z =   -1.000 mm,
	W =-180.000 deg,	P =   0.000 deg,	R =    90.000 deg
};
P[5331]{
   GP1:
	UF : 1, UT : 3,		CONFIG : 'N U T, 0, 0, 0',
	X =  34.000  mm,	Y =  100.000  mm,	Z =   15.000 mm,
	W =-180.000 deg,	P =   0.000 deg,	R =    90.000 deg
};
P[5332]{
   GP1:
	UF : 1, UT : 3,		CONFIG : 'N U T, 0, 0, 0',
	X =  37.000  mm,	Y =  100.000  mm,	Z =   15.000 mm,
	W =-180.000 deg,	P =   0.000 deg,	R =    90.000 deg
};
P[5333]{
   GP1:
	UF : 1, UT : 3,		CONFIG : 'N U T, 0, 0, 0',
	X =  37.000  mm,	Y =  100.000  mm,	Z =   -1.000 mm,
	W =-180.000 deg,	P =   0.000 deg,	R =    90.000 deg
};
P[5334]{
   GP1:
	UF : 1, UT : 3,		CONFIG : 'N U T, 0, 0, 0',
	X =  37.000  mm,	Y =  100.000  mm,	Z =   15.000 mm,
	W =-180.000 deg,	P =   0.000 deg,	R =    90.000 deg
};
P[5359]{
   GP1:
	UF : 1, UT : 3,		CONFIG : 'N U T, 0, 0, 0',
	X =  64.000  mm,	Y =  100.000  mm,	Z =   15.000 mm,
	W =-180.000 deg,	P =   0.000 deg,	R =    90.000 deg
};
P[5360]{
   GP1:
	UF : 1, UT : 3,		CONFIG : 'N U T, 0, 0, 0',
	X =  64.000  mm,	Y =  100.000  mm,	Z =   -1.000 mm,
	W =-180.000 deg,	P =   0.000 deg,	R =    90.000 deg
};
P[5361]{
   GP1:
	UF : 1, UT : 3,		CONFIG : 'N U T, 0, 0, 0',
	X =  64.000  mm,	Y =  100.000  mm,	Z =   15.000 mm,
	W =-180.000 deg,	P =   0.000 deg,	R =    90.000 deg
};
P[5362]{
   GP1:
	UF : 1, UT : 3,		CONFIG : 'N U T, 0, 0, 0',
	X =  67.000  mm,	Y =  100.000  mm,	Z =   15.000 mm,
	W =-180.000 deg,	P =   0.000 deg,	R =    90.000 deg
};
P[5363]{
   GP1:
	UF : 1, UT : 3,		CONFIG : 'N U T, 0, 0, 0',
	X =  67.000  mm,	Y =  100.000  mm,	Z =   -1.000 mm,
	W =-180.000 deg,	P =   0.000 deg,	R =    90.000 deg
};
P[5364]{
   GP1:
	UF : 1, UT : 3,		CONFIG : 'N U T, 0, 0, 0',
	X =  67.000  mm,	Y =  100.000  mm,	Z =   15.000 mm,
	W =-180.000 deg,	P =   0.000 deg,	R =    90.000 deg
};
P[5365]{
   GP1:
	UF : 1, UT : 3,		CONFIG : 'N U T, 0, 0, 0',
	X =  70.000  mm,	Y =  100.000  mm,	Z =   15.000 mm,
	W =-180.000 deg,	P =   0.000 deg,	R =    90.000 deg
};
P[5366]{
   GP1:
	UF : 1, UT : 3,		CONFIG : 'N U T, 0, 0, 0',
	X =  70.000  mm,	Y =  100.000  mm,	Z =   -1.000 mm,
	W =-180.000 deg,	P =   0.000 deg,	R =    90.000 deg
};
P[5367]{
   GP1:
	UF : 1, UT : 3,		CONFIG : 'N U T, 0, 0, 0',
	X =  70.000  mm,	Y =  100.000  mm,	Z =   15.000 mm,
	W =-180.000 deg,	P =   0.000 deg,	R =    90.000 deg
};
P[5368]{
   GP1:
	UF : 1, UT : 3,		CONFIG : 'N U T, 0, 0, 0',
	X =  73.000  mm,	Y =  100.000  mm,	Z =   15.000 mm,
	W =-180.000 deg,	P =   0.000 deg,	R =    90.000 deg
};
P[5369]{
   GP1:
	UF : 1, UT : 3,		CONFIG : 'N U T, 0, 0, 0',
	X =  73.000  mm,	Y =  100.000  mm,	Z =   -1.000 mm,
	W =-180.000 deg,	P =   0.000 deg,	R =    90.000 deg
};
P[5370]{
   GP1:
	UF : 1, UT : 3,		CONFIG : 'N U T, 0, 0, 0',
	X =  73.000  mm,	Y =  100.000  mm,	Z =   15.000 mm,
	W =-180.000 deg,	P =   0.000 deg,	R =    90.000 deg
};
P[5371]{
   GP1:
	UF : 1, UT : 3,		CONFIG : 'N U T, 0, 0, 0',
	X =  76.000  mm,	Y =  100.000  mm,	Z =   15.000 mm,
	W =-180.000 deg,	P =   0.000 deg,	R =    90.000 deg
};
P[5372]{
   GP1:
	UF : 1, UT : 3,		CONFIG : 'N U T, 0, 0, 0',
	X =  76.000  mm,	Y =  100.000  mm,	Z =   -1.000 mm,
	W =-180.000 deg,	P =   0.000 deg,	R =    90.000 deg
};
P[5373]{
   GP1:
	UF : 1, UT : 3,		CONFIG : 'N U T, 0, 0, 0',
	X =  76.000  mm,	Y =  100.000  mm,	Z =   15.000 mm,
	W =-180.000 deg,	P =   0.000 deg,	R =    90.000 deg
};
P[5374]{
   GP1:
	UF : 1, UT : 3,		CONFIG : 'N U T, 0, 0, 0',
	X =  79.000  mm,	Y =  100.000  mm,	Z =   15.000 mm,
	W =-180.000 deg,	P =   0.000 deg,	R =    90.000 deg
};
P[5375]{
   GP1:
	UF : 1, UT : 3,		CONFIG : 'N U T, 0, 0, 0',
	X =  79.000  mm,	Y =  100.000  mm,	Z =   -1.000 mm,
	W =-180.000 deg,	P =   0.000 deg,	R =    90.000 deg
};
P[5376]{
   GP1:
	UF : 1, UT : 3,		CONFIG : 'N U T, 0, 0, 0',
	X =  79.000  mm,	Y =  100.000  mm,	Z =   15.000 mm,
	W =-180.000 deg,	P =   0.000 deg,	R =    90.000 deg
};
P[5377]{
   GP1:
	UF : 1, UT : 3,		CONFIG : 'N U T, 0, 0, 0',
	X =  82.000  mm,	Y =  100.000  mm,	Z =   15.000 mm,
	W =-180.000 deg,	P =   0.000 deg,	R =    90.000 deg
};
P[5378]{
   GP1:
	UF : 1, UT : 3,		CONFIG : 'N U T, 0, 0, 0',
	X =  82.000  mm,	Y =  100.000  mm,	Z =   -1.000 mm,
	W =-180.000 deg,	P =   0.000 deg,	R =    90.000 deg
};
P[5379]{
   GP1:
	UF : 1, UT : 3,		CONFIG : 'N U T, 0, 0, 0',
	X =  82.000  mm,	Y =  100.000  mm,	Z =   15.000 mm,
	W =-180.000 deg,	P =   0.000 deg,	R =    90.000 deg
};
P[5380]{
   GP1:
	UF : 1, UT : 3,		CONFIG : 'N U T, 0, 0, 0',
	X =  85.000  mm,	Y =  100.000  mm,	Z =   15.000 mm,
	W =-180.000 deg,	P =   0.000 deg,	R =    90.000 deg
};
P[5381]{
   GP1:
	UF : 1, UT : 3,		CONFIG : 'N U T, 0, 0, 0',
	X =  85.000  mm,	Y =  100.000  mm,	Z =   -1.000 mm,
	W =-180.000 deg,	P =   0.000 deg,	R =    90.000 deg
};
P[5382]{
   GP1:
	UF : 1, UT : 3,		CONFIG : 'N U T, 0, 0, 0',
	X =  85.000  mm,	Y =  100.000  mm,	Z =   15.000 mm,
	W =-180.000 deg,	P =   0.000 deg,	R =    90.000 deg
};
P[5383]{
   GP1:
	UF : 1, UT : 3,		CONFIG : 'N U T, 0, 0, 0',
	X =  88.000  mm,	Y =  100.000  mm,	Z =   15.000 mm,
	W =-180.000 deg,	P =   0.000 deg,	R =    90.000 deg
};
P[5384]{
   GP1:
	UF : 1, UT : 3,		CONFIG : 'N U T, 0, 0, 0',
	X =  88.000  mm,	Y =  100.000  mm,	Z =   -1.000 mm,
	W =-180.000 deg,	P =   0.000 deg,	R =    90.000 deg
};
P[5385]{
   GP1:
	UF : 1, UT : 3,		CONFIG : 'N U T, 0, 0, 0',
	X =  88.000  mm,	Y =  100.000  mm,	Z =   15.000 mm,
	W =-180.000 deg,	P =   0.000 deg,	R =    90.000 deg
};
P[5416]{
   GP1:
	UF : 1, UT : 3,		CONFIG : 'N U T, 0, 0, 0',
	X =  121.000  mm,	Y =  100.000  mm,	Z =   15.000 mm,
	W =-180.000 deg,	P =   0.000 deg,	R =    90.000 deg
};
P[5417]{
   GP1:
	UF : 1, UT : 3,		CONFIG : 'N U T, 0, 0, 0',
	X =  121.000  mm,	Y =  100.000  mm,	Z =   -1.000 mm,
	W =-180.000 deg,	P =   0.000 deg,	R =    90.000 deg
};
P[5418]{
   GP1:
	UF : 1, UT : 3,		CONFIG : 'N U T, 0, 0, 0',
	X =  121.000  mm,	Y =  100.000  mm,	Z =   15.000 mm,
	W =-180.000 deg,	P =   0.000 deg,	R =    90.000 deg
};
P[5419]{
   GP1:
	UF : 1, UT : 3,		CONFIG : 'N U T, 0, 0, 0',
	X =  124.000  mm,	Y =  100.000  mm,	Z =   15.000 mm,
	W =-180.000 deg,	P =   0.000 deg,	R =    90.000 deg
};
P[5420]{
   GP1:
	UF : 1, UT : 3,		CONFIG : 'N U T, 0, 0, 0',
	X =  124.000  mm,	Y =  100.000  mm,	Z =   -1.000 mm,
	W =-180.000 deg,	P =   0.000 deg,	R =    90.000 deg
};
P[5421]{
   GP1:
	UF : 1, UT : 3,		CONFIG : 'N U T, 0, 0, 0',
	X =  124.000  mm,	Y =  100.000  mm,	Z =   15.000 mm,
	W =-180.000 deg,	P =   0.000 deg,	R =    90.000 deg
};
P[5440]{
   GP1:
	UF : 1, UT : 3,		CONFIG : 'N U T, 0, 0, 0',
	X =  145.000  mm,	Y =  100.000  mm,	Z =   15.000 mm,
	W =-180.000 deg,	P =   0.000 deg,	R =    90.000 deg
};
P[5441]{
   GP1:
	UF : 1, UT : 3,		CONFIG : 'N U T, 0, 0, 0',
	X =  145.000  mm,	Y =  100.000  mm,	Z =   -1.000 mm,
	W =-180.000 deg,	P =   0.000 deg,	R =    90.000 deg
};
P[5442]{
   GP1:
	UF : 1, UT : 3,		CONFIG : 'N U T, 0, 0, 0',
	X =  145.000  mm,	Y =  100.000  mm,	Z =   15.000 mm,
	W =-180.000 deg,	P =   0.000 deg,	R =    90.000 deg
};
P[5443]{
   GP1:
	UF : 1, UT : 3,		CONFIG : 'N U T, 0, 0, 0',
	X =  148.000  mm,	Y =  100.000  mm,	Z =   15.000 mm,
	W =-180.000 deg,	P =   0.000 deg,	R =    90.000 deg
};
P[5444]{
   GP1:
	UF : 1, UT : 3,		CONFIG : 'N U T, 0, 0, 0',
	X =  148.000  mm,	Y =  100.000  mm,	Z =   -1.000 mm,
	W =-180.000 deg,	P =   0.000 deg,	R =    90.000 deg
};
P[5445]{
   GP1:
	UF : 1, UT : 3,		CONFIG : 'N U T, 0, 0, 0',
	X =  148.000  mm,	Y =  100.000  mm,	Z =   15.000 mm,
	W =-180.000 deg,	P =   0.000 deg,	R =    90.000 deg
};
P[5485]{
   GP1:
	UF : 1, UT : 3,		CONFIG : 'N U T, 0, 0, 0',
	X =  22.000  mm,	Y =  103.000  mm,	Z =   15.000 mm,
	W =-180.000 deg,	P =   0.000 deg,	R =    90.000 deg
};
P[5486]{
   GP1:
	UF : 1, UT : 3,		CONFIG : 'N U T, 0, 0, 0',
	X =  22.000  mm,	Y =  103.000  mm,	Z =   -1.000 mm,
	W =-180.000 deg,	P =   0.000 deg,	R =    90.000 deg
};
P[5487]{
   GP1:
	UF : 1, UT : 3,		CONFIG : 'N U T, 0, 0, 0',
	X =  22.000  mm,	Y =  103.000  mm,	Z =   15.000 mm,
	W =-180.000 deg,	P =   0.000 deg,	R =    90.000 deg
};
P[5488]{
   GP1:
	UF : 1, UT : 3,		CONFIG : 'N U T, 0, 0, 0',
	X =  25.000  mm,	Y =  103.000  mm,	Z =   15.000 mm,
	W =-180.000 deg,	P =   0.000 deg,	R =    90.000 deg
};
P[5489]{
   GP1:
	UF : 1, UT : 3,		CONFIG : 'N U T, 0, 0, 0',
	X =  25.000  mm,	Y =  103.000  mm,	Z =   -1.000 mm,
	W =-180.000 deg,	P =   0.000 deg,	R =    90.000 deg
};
P[5490]{
   GP1:
	UF : 1, UT : 3,		CONFIG : 'N U T, 0, 0, 0',
	X =  25.000  mm,	Y =  103.000  mm,	Z =   15.000 mm,
	W =-180.000 deg,	P =   0.000 deg,	R =    90.000 deg
};
P[5518]{
   GP1:
	UF : 1, UT : 3,		CONFIG : 'N U T, 0, 0, 0',
	X =  55.000  mm,	Y =  103.000  mm,	Z =   15.000 mm,
	W =-180.000 deg,	P =   0.000 deg,	R =    90.000 deg
};
P[5519]{
   GP1:
	UF : 1, UT : 3,		CONFIG : 'N U T, 0, 0, 0',
	X =  55.000  mm,	Y =  103.000  mm,	Z =   -1.000 mm,
	W =-180.000 deg,	P =   0.000 deg,	R =    90.000 deg
};
P[5520]{
   GP1:
	UF : 1, UT : 3,		CONFIG : 'N U T, 0, 0, 0',
	X =  55.000  mm,	Y =  103.000  mm,	Z =   15.000 mm,
	W =-180.000 deg,	P =   0.000 deg,	R =    90.000 deg
};
P[5596]{
   GP1:
	UF : 1, UT : 3,		CONFIG : 'N U T, 0, 0, 0',
	X =  133.000  mm,	Y =  103.000  mm,	Z =   15.000 mm,
	W =-180.000 deg,	P =   0.000 deg,	R =    90.000 deg
};
P[5597]{
   GP1:
	UF : 1, UT : 3,		CONFIG : 'N U T, 0, 0, 0',
	X =  133.000  mm,	Y =  103.000  mm,	Z =   -1.000 mm,
	W =-180.000 deg,	P =   0.000 deg,	R =    90.000 deg
};
P[5598]{
   GP1:
	UF : 1, UT : 3,		CONFIG : 'N U T, 0, 0, 0',
	X =  133.000  mm,	Y =  103.000  mm,	Z =   15.000 mm,
	W =-180.000 deg,	P =   0.000 deg,	R =    90.000 deg
};
P[5656]{
   GP1:
	UF : 1, UT : 3,		CONFIG : 'N U T, 0, 0, 0',
	X =  22.000  mm,	Y =  106.000  mm,	Z =   15.000 mm,
	W =-180.000 deg,	P =   0.000 deg,	R =    90.000 deg
};
P[5657]{
   GP1:
	UF : 1, UT : 3,		CONFIG : 'N U T, 0, 0, 0',
	X =  22.000  mm,	Y =  106.000  mm,	Z =   -1.000 mm,
	W =-180.000 deg,	P =   0.000 deg,	R =    90.000 deg
};
P[5658]{
   GP1:
	UF : 1, UT : 3,		CONFIG : 'N U T, 0, 0, 0',
	X =  22.000  mm,	Y =  106.000  mm,	Z =   15.000 mm,
	W =-180.000 deg,	P =   0.000 deg,	R =    90.000 deg
};
P[5662]{
   GP1:
	UF : 1, UT : 3,		CONFIG : 'N U T, 0, 0, 0',
	X =  28.000  mm,	Y =  106.000  mm,	Z =   15.000 mm,
	W =-180.000 deg,	P =   0.000 deg,	R =    90.000 deg
};
P[5663]{
   GP1:
	UF : 1, UT : 3,		CONFIG : 'N U T, 0, 0, 0',
	X =  28.000  mm,	Y =  106.000  mm,	Z =   -1.000 mm,
	W =-180.000 deg,	P =   0.000 deg,	R =    90.000 deg
};
P[5664]{
   GP1:
	UF : 1, UT : 3,		CONFIG : 'N U T, 0, 0, 0',
	X =  28.000  mm,	Y =  106.000  mm,	Z =   15.000 mm,
	W =-180.000 deg,	P =   0.000 deg,	R =    90.000 deg
};
P[5665]{
   GP1:
	UF : 1, UT : 3,		CONFIG : 'N U T, 0, 0, 0',
	X =  31.000  mm,	Y =  106.000  mm,	Z =   15.000 mm,
	W =-180.000 deg,	P =   0.000 deg,	R =    90.000 deg
};
P[5666]{
   GP1:
	UF : 1, UT : 3,		CONFIG : 'N U T, 0, 0, 0',
	X =  31.000  mm,	Y =  106.000  mm,	Z =   -1.000 mm,
	W =-180.000 deg,	P =   0.000 deg,	R =    90.000 deg
};
P[5667]{
   GP1:
	UF : 1, UT : 3,		CONFIG : 'N U T, 0, 0, 0',
	X =  31.000  mm,	Y =  106.000  mm,	Z =   15.000 mm,
	W =-180.000 deg,	P =   0.000 deg,	R =    90.000 deg
};
P[5677]{
   GP1:
	UF : 1, UT : 3,		CONFIG : 'N U T, 0, 0, 0',
	X =  43.000  mm,	Y =  106.000  mm,	Z =   15.000 mm,
	W =-180.000 deg,	P =   0.000 deg,	R =    90.000 deg
};
P[5678]{
   GP1:
	UF : 1, UT : 3,		CONFIG : 'N U T, 0, 0, 0',
	X =  43.000  mm,	Y =  106.000  mm,	Z =   -1.000 mm,
	W =-180.000 deg,	P =   0.000 deg,	R =    90.000 deg
};
P[5679]{
   GP1:
	UF : 1, UT : 3,		CONFIG : 'N U T, 0, 0, 0',
	X =  43.000  mm,	Y =  106.000  mm,	Z =   15.000 mm,
	W =-180.000 deg,	P =   0.000 deg,	R =    90.000 deg
};
P[5734]{
   GP1:
	UF : 1, UT : 3,		CONFIG : 'N U T, 0, 0, 0',
	X =  142.000  mm,	Y =  106.000  mm,	Z =   15.000 mm,
	W =-180.000 deg,	P =   0.000 deg,	R =    90.000 deg
};
P[5735]{
   GP1:
	UF : 1, UT : 3,		CONFIG : 'N U T, 0, 0, 0',
	X =  142.000  mm,	Y =  106.000  mm,	Z =   -1.000 mm,
	W =-180.000 deg,	P =   0.000 deg,	R =    90.000 deg
};
P[5736]{
   GP1:
	UF : 1, UT : 3,		CONFIG : 'N U T, 0, 0, 0',
	X =  142.000  mm,	Y =  106.000  mm,	Z =   15.000 mm,
	W =-180.000 deg,	P =   0.000 deg,	R =    90.000 deg
};
P[5740]{
   GP1:
	UF : 1, UT : 3,		CONFIG : 'N U T, 0, 0, 0',
	X =  160.000  mm,	Y =  106.000  mm,	Z =   15.000 mm,
	W =-180.000 deg,	P =   0.000 deg,	R =    90.000 deg
};
P[5741]{
   GP1:
	UF : 1, UT : 3,		CONFIG : 'N U T, 0, 0, 0',
	X =  160.000  mm,	Y =  106.000  mm,	Z =   -1.000 mm,
	W =-180.000 deg,	P =   0.000 deg,	R =    90.000 deg
};
P[5742]{
   GP1:
	UF : 1, UT : 3,		CONFIG : 'N U T, 0, 0, 0',
	X =  160.000  mm,	Y =  106.000  mm,	Z =   15.000 mm,
	W =-180.000 deg,	P =   0.000 deg,	R =    90.000 deg
};
P[5779]{
   GP1:
	UF : 1, UT : 3,		CONFIG : 'N U T, 0, 0, 0',
	X =  22.000  mm,	Y =  109.000  mm,	Z =   15.000 mm,
	W =-180.000 deg,	P =   0.000 deg,	R =    90.000 deg
};
P[5780]{
   GP1:
	UF : 1, UT : 3,		CONFIG : 'N U T, 0, 0, 0',
	X =  22.000  mm,	Y =  109.000  mm,	Z =   -1.000 mm,
	W =-180.000 deg,	P =   0.000 deg,	R =    90.000 deg
};
P[5781]{
   GP1:
	UF : 1, UT : 3,		CONFIG : 'N U T, 0, 0, 0',
	X =  22.000  mm,	Y =  109.000  mm,	Z =   15.000 mm,
	W =-180.000 deg,	P =   0.000 deg,	R =    90.000 deg
};
P[5782]{
   GP1:
	UF : 1, UT : 3,		CONFIG : 'N U T, 0, 0, 0',
	X =  25.000  mm,	Y =  109.000  mm,	Z =   15.000 mm,
	W =-180.000 deg,	P =   0.000 deg,	R =    90.000 deg
};
P[5783]{
   GP1:
	UF : 1, UT : 3,		CONFIG : 'N U T, 0, 0, 0',
	X =  25.000  mm,	Y =  109.000  mm,	Z =   -1.000 mm,
	W =-180.000 deg,	P =   0.000 deg,	R =    90.000 deg
};
P[5784]{
   GP1:
	UF : 1, UT : 3,		CONFIG : 'N U T, 0, 0, 0',
	X =  25.000  mm,	Y =  109.000  mm,	Z =   15.000 mm,
	W =-180.000 deg,	P =   0.000 deg,	R =    90.000 deg
};
P[5785]{
   GP1:
	UF : 1, UT : 3,		CONFIG : 'N U T, 0, 0, 0',
	X =  28.000  mm,	Y =  109.000  mm,	Z =   15.000 mm,
	W =-180.000 deg,	P =   0.000 deg,	R =    90.000 deg
};
P[5786]{
   GP1:
	UF : 1, UT : 3,		CONFIG : 'N U T, 0, 0, 0',
	X =  28.000  mm,	Y =  109.000  mm,	Z =   -1.000 mm,
	W =-180.000 deg,	P =   0.000 deg,	R =    90.000 deg
};
P[5787]{
   GP1:
	UF : 1, UT : 3,		CONFIG : 'N U T, 0, 0, 0',
	X =  28.000  mm,	Y =  109.000  mm,	Z =   15.000 mm,
	W =-180.000 deg,	P =   0.000 deg,	R =    90.000 deg
};
P[5812]{
   GP1:
	UF : 1, UT : 3,		CONFIG : 'N U T, 0, 0, 0',
	X =  55.000  mm,	Y =  109.000  mm,	Z =   15.000 mm,
	W =-180.000 deg,	P =   0.000 deg,	R =    90.000 deg
};
P[5813]{
   GP1:
	UF : 1, UT : 3,		CONFIG : 'N U T, 0, 0, 0',
	X =  55.000  mm,	Y =  109.000  mm,	Z =   -1.000 mm,
	W =-180.000 deg,	P =   0.000 deg,	R =    90.000 deg
};
P[5814]{
   GP1:
	UF : 1, UT : 3,		CONFIG : 'N U T, 0, 0, 0',
	X =  55.000  mm,	Y =  109.000  mm,	Z =   15.000 mm,
	W =-180.000 deg,	P =   0.000 deg,	R =    90.000 deg
};
P[5833]{
   GP1:
	UF : 1, UT : 3,		CONFIG : 'N U T, 0, 0, 0',
	X =  127.000  mm,	Y =  109.000  mm,	Z =   15.000 mm,
	W =-180.000 deg,	P =   0.000 deg,	R =    90.000 deg
};
P[5834]{
   GP1:
	UF : 1, UT : 3,		CONFIG : 'N U T, 0, 0, 0',
	X =  127.000  mm,	Y =  109.000  mm,	Z =   -1.000 mm,
	W =-180.000 deg,	P =   0.000 deg,	R =    90.000 deg
};
P[5835]{
   GP1:
	UF : 1, UT : 3,		CONFIG : 'N U T, 0, 0, 0',
	X =  127.000  mm,	Y =  109.000  mm,	Z =   15.000 mm,
	W =-180.000 deg,	P =   0.000 deg,	R =    90.000 deg
};
P[5836]{
   GP1:
	UF : 1, UT : 3,		CONFIG : 'N U T, 0, 0, 0',
	X =  130.000  mm,	Y =  109.000  mm,	Z =   15.000 mm,
	W =-180.000 deg,	P =   0.000 deg,	R =    90.000 deg
};
P[5837]{
   GP1:
	UF : 1, UT : 3,		CONFIG : 'N U T, 0, 0, 0',
	X =  130.000  mm,	Y =  109.000  mm,	Z =   -1.000 mm,
	W =-180.000 deg,	P =   0.000 deg,	R =    90.000 deg
};
P[5838]{
   GP1:
	UF : 1, UT : 3,		CONFIG : 'N U T, 0, 0, 0',
	X =  130.000  mm,	Y =  109.000  mm,	Z =   15.000 mm,
	W =-180.000 deg,	P =   0.000 deg,	R =    90.000 deg
};
P[5845]{
   GP1:
	UF : 1, UT : 3,		CONFIG : 'N U T, 0, 0, 0',
	X =  139.000  mm,	Y =  109.000  mm,	Z =   15.000 mm,
	W =-180.000 deg,	P =   0.000 deg,	R =    90.000 deg
};
P[5846]{
   GP1:
	UF : 1, UT : 3,		CONFIG : 'N U T, 0, 0, 0',
	X =  139.000  mm,	Y =  109.000  mm,	Z =   -1.000 mm,
	W =-180.000 deg,	P =   0.000 deg,	R =    90.000 deg
};
P[5847]{
   GP1:
	UF : 1, UT : 3,		CONFIG : 'N U T, 0, 0, 0',
	X =  139.000  mm,	Y =  109.000  mm,	Z =   15.000 mm,
	W =-180.000 deg,	P =   0.000 deg,	R =    90.000 deg
};
P[5881]{
   GP1:
	UF : 1, UT : 3,		CONFIG : 'N U T, 0, 0, 0',
	X =  19.000  mm,	Y =  112.000  mm,	Z =   15.000 mm,
	W =-180.000 deg,	P =   0.000 deg,	R =    90.000 deg
};
P[5882]{
   GP1:
	UF : 1, UT : 3,		CONFIG : 'N U T, 0, 0, 0',
	X =  19.000  mm,	Y =  112.000  mm,	Z =   -1.000 mm,
	W =-180.000 deg,	P =   0.000 deg,	R =    90.000 deg
};
P[5883]{
   GP1:
	UF : 1, UT : 3,		CONFIG : 'N U T, 0, 0, 0',
	X =  19.000  mm,	Y =  112.000  mm,	Z =   15.000 mm,
	W =-180.000 deg,	P =   0.000 deg,	R =    90.000 deg
};
P[5884]{
   GP1:
	UF : 1, UT : 3,		CONFIG : 'N U T, 0, 0, 0',
	X =  22.000  mm,	Y =  112.000  mm,	Z =   15.000 mm,
	W =-180.000 deg,	P =   0.000 deg,	R =    90.000 deg
};
P[5885]{
   GP1:
	UF : 1, UT : 3,		CONFIG : 'N U T, 0, 0, 0',
	X =  22.000  mm,	Y =  112.000  mm,	Z =   -1.000 mm,
	W =-180.000 deg,	P =   0.000 deg,	R =    90.000 deg
};
P[5886]{
   GP1:
	UF : 1, UT : 3,		CONFIG : 'N U T, 0, 0, 0',
	X =  22.000  mm,	Y =  112.000  mm,	Z =   15.000 mm,
	W =-180.000 deg,	P =   0.000 deg,	R =    90.000 deg
};
P[5914]{
   GP1:
	UF : 1, UT : 3,		CONFIG : 'N U T, 0, 0, 0',
	X =  52.000  mm,	Y =  112.000  mm,	Z =   15.000 mm,
	W =-180.000 deg,	P =   0.000 deg,	R =    90.000 deg
};
P[5915]{
   GP1:
	UF : 1, UT : 3,		CONFIG : 'N U T, 0, 0, 0',
	X =  52.000  mm,	Y =  112.000  mm,	Z =   -1.000 mm,
	W =-180.000 deg,	P =   0.000 deg,	R =    90.000 deg
};
P[5916]{
   GP1:
	UF : 1, UT : 3,		CONFIG : 'N U T, 0, 0, 0',
	X =  52.000  mm,	Y =  112.000  mm,	Z =   15.000 mm,
	W =-180.000 deg,	P =   0.000 deg,	R =    90.000 deg
};
P[5917]{
   GP1:
	UF : 1, UT : 3,		CONFIG : 'N U T, 0, 0, 0',
	X =  55.000  mm,	Y =  112.000  mm,	Z =   15.000 mm,
	W =-180.000 deg,	P =   0.000 deg,	R =    90.000 deg
};
P[5918]{
   GP1:
	UF : 1, UT : 3,		CONFIG : 'N U T, 0, 0, 0',
	X =  55.000  mm,	Y =  112.000  mm,	Z =   -1.000 mm,
	W =-180.000 deg,	P =   0.000 deg,	R =    90.000 deg
};
P[5919]{
   GP1:
	UF : 1, UT : 3,		CONFIG : 'N U T, 0, 0, 0',
	X =  55.000  mm,	Y =  112.000  mm,	Z =   15.000 mm,
	W =-180.000 deg,	P =   0.000 deg,	R =    90.000 deg
};
P[5929]{
   GP1:
	UF : 1, UT : 3,		CONFIG : 'N U T, 0, 0, 0',
	X =  124.000  mm,	Y =  112.000  mm,	Z =   15.000 mm,
	W =-180.000 deg,	P =   0.000 deg,	R =    90.000 deg
};
P[5930]{
   GP1:
	UF : 1, UT : 3,		CONFIG : 'N U T, 0, 0, 0',
	X =  124.000  mm,	Y =  112.000  mm,	Z =   -1.000 mm,
	W =-180.000 deg,	P =   0.000 deg,	R =    90.000 deg
};
P[5931]{
   GP1:
	UF : 1, UT : 3,		CONFIG : 'N U T, 0, 0, 0',
	X =  124.000  mm,	Y =  112.000  mm,	Z =   15.000 mm,
	W =-180.000 deg,	P =   0.000 deg,	R =    90.000 deg
};
P[5968]{
   GP1:
	UF : 1, UT : 3,		CONFIG : 'N U T, 0, 0, 0',
	X =  19.000  mm,	Y =  115.000  mm,	Z =   15.000 mm,
	W =-180.000 deg,	P =   0.000 deg,	R =    90.000 deg
};
P[5969]{
   GP1:
	UF : 1, UT : 3,		CONFIG : 'N U T, 0, 0, 0',
	X =  19.000  mm,	Y =  115.000  mm,	Z =   -1.000 mm,
	W =-180.000 deg,	P =   0.000 deg,	R =    90.000 deg
};
P[5970]{
   GP1:
	UF : 1, UT : 3,		CONFIG : 'N U T, 0, 0, 0',
	X =  19.000  mm,	Y =  115.000  mm,	Z =   15.000 mm,
	W =-180.000 deg,	P =   0.000 deg,	R =    90.000 deg
};
P[5971]{
   GP1:
	UF : 1, UT : 3,		CONFIG : 'N U T, 0, 0, 0',
	X =  22.000  mm,	Y =  115.000  mm,	Z =   15.000 mm,
	W =-180.000 deg,	P =   0.000 deg,	R =    90.000 deg
};
P[5972]{
   GP1:
	UF : 1, UT : 3,		CONFIG : 'N U T, 0, 0, 0',
	X =  22.000  mm,	Y =  115.000  mm,	Z =   -1.000 mm,
	W =-180.000 deg,	P =   0.000 deg,	R =    90.000 deg
};
P[5973]{
   GP1:
	UF : 1, UT : 3,		CONFIG : 'N U T, 0, 0, 0',
	X =  22.000  mm,	Y =  115.000  mm,	Z =   15.000 mm,
	W =-180.000 deg,	P =   0.000 deg,	R =    90.000 deg
};
P[6034]{
   GP1:
	UF : 1, UT : 3,		CONFIG : 'N U T, 0, 0, 0',
	X =  142.000  mm,	Y =  115.000  mm,	Z =   15.000 mm,
	W =-180.000 deg,	P =   0.000 deg,	R =    90.000 deg
};
P[6035]{
   GP1:
	UF : 1, UT : 3,		CONFIG : 'N U T, 0, 0, 0',
	X =  142.000  mm,	Y =  115.000  mm,	Z =   -1.000 mm,
	W =-180.000 deg,	P =   0.000 deg,	R =    90.000 deg
};
P[6036]{
   GP1:
	UF : 1, UT : 3,		CONFIG : 'N U T, 0, 0, 0',
	X =  142.000  mm,	Y =  115.000  mm,	Z =   15.000 mm,
	W =-180.000 deg,	P =   0.000 deg,	R =    90.000 deg
};
P[6064]{
   GP1:
	UF : 1, UT : 3,		CONFIG : 'N U T, 0, 0, 0',
	X =  22.000  mm,	Y =  118.000  mm,	Z =   15.000 mm,
	W =-180.000 deg,	P =   0.000 deg,	R =    90.000 deg
};
P[6065]{
   GP1:
	UF : 1, UT : 3,		CONFIG : 'N U T, 0, 0, 0',
	X =  22.000  mm,	Y =  118.000  mm,	Z =   -1.000 mm,
	W =-180.000 deg,	P =   0.000 deg,	R =    90.000 deg
};
P[6066]{
   GP1:
	UF : 1, UT : 3,		CONFIG : 'N U T, 0, 0, 0',
	X =  22.000  mm,	Y =  118.000  mm,	Z =   15.000 mm,
	W =-180.000 deg,	P =   0.000 deg,	R =    90.000 deg
};
P[6073]{
   GP1:
	UF : 1, UT : 3,		CONFIG : 'N U T, 0, 0, 0',
	X =  31.000  mm,	Y =  118.000  mm,	Z =   15.000 mm,
	W =-180.000 deg,	P =   0.000 deg,	R =    90.000 deg
};
P[6074]{
   GP1:
	UF : 1, UT : 3,		CONFIG : 'N U T, 0, 0, 0',
	X =  31.000  mm,	Y =  118.000  mm,	Z =   -1.000 mm,
	W =-180.000 deg,	P =   0.000 deg,	R =    90.000 deg
};
P[6075]{
   GP1:
	UF : 1, UT : 3,		CONFIG : 'N U T, 0, 0, 0',
	X =  31.000  mm,	Y =  118.000  mm,	Z =   15.000 mm,
	W =-180.000 deg,	P =   0.000 deg,	R =    90.000 deg
};
P[6163]{
   GP1:
	UF : 1, UT : 3,		CONFIG : 'N U T, 0, 0, 0',
	X =  19.000  mm,	Y =  121.000  mm,	Z =   15.000 mm,
	W =-180.000 deg,	P =   0.000 deg,	R =    90.000 deg
};
P[6164]{
   GP1:
	UF : 1, UT : 3,		CONFIG : 'N U T, 0, 0, 0',
	X =  19.000  mm,	Y =  121.000  mm,	Z =   -1.000 mm,
	W =-180.000 deg,	P =   0.000 deg,	R =    90.000 deg
};
P[6165]{
   GP1:
	UF : 1, UT : 3,		CONFIG : 'N U T, 0, 0, 0',
	X =  19.000  mm,	Y =  121.000  mm,	Z =   15.000 mm,
	W =-180.000 deg,	P =   0.000 deg,	R =    90.000 deg
};
P[6166]{
   GP1:
	UF : 1, UT : 3,		CONFIG : 'N U T, 0, 0, 0',
	X =  22.000  mm,	Y =  121.000  mm,	Z =   15.000 mm,
	W =-180.000 deg,	P =   0.000 deg,	R =    90.000 deg
};
P[6167]{
   GP1:
	UF : 1, UT : 3,		CONFIG : 'N U T, 0, 0, 0',
	X =  22.000  mm,	Y =  121.000  mm,	Z =   -1.000 mm,
	W =-180.000 deg,	P =   0.000 deg,	R =    90.000 deg
};
P[6168]{
   GP1:
	UF : 1, UT : 3,		CONFIG : 'N U T, 0, 0, 0',
	X =  22.000  mm,	Y =  121.000  mm,	Z =   15.000 mm,
	W =-180.000 deg,	P =   0.000 deg,	R =    90.000 deg
};
P[6169]{
   GP1:
	UF : 1, UT : 3,		CONFIG : 'N U T, 0, 0, 0',
	X =  25.000  mm,	Y =  121.000  mm,	Z =   15.000 mm,
	W =-180.000 deg,	P =   0.000 deg,	R =    90.000 deg
};
P[6170]{
   GP1:
	UF : 1, UT : 3,		CONFIG : 'N U T, 0, 0, 0',
	X =  25.000  mm,	Y =  121.000  mm,	Z =   -1.000 mm,
	W =-180.000 deg,	P =   0.000 deg,	R =    90.000 deg
};
P[6171]{
   GP1:
	UF : 1, UT : 3,		CONFIG : 'N U T, 0, 0, 0',
	X =  25.000  mm,	Y =  121.000  mm,	Z =   15.000 mm,
	W =-180.000 deg,	P =   0.000 deg,	R =    90.000 deg
};
P[6175]{
   GP1:
	UF : 1, UT : 3,		CONFIG : 'N U T, 0, 0, 0',
	X =  31.000  mm,	Y =  121.000  mm,	Z =   15.000 mm,
	W =-180.000 deg,	P =   0.000 deg,	R =    90.000 deg
};
P[6176]{
   GP1:
	UF : 1, UT : 3,		CONFIG : 'N U T, 0, 0, 0',
	X =  31.000  mm,	Y =  121.000  mm,	Z =   -1.000 mm,
	W =-180.000 deg,	P =   0.000 deg,	R =    90.000 deg
};
P[6177]{
   GP1:
	UF : 1, UT : 3,		CONFIG : 'N U T, 0, 0, 0',
	X =  31.000  mm,	Y =  121.000  mm,	Z =   15.000 mm,
	W =-180.000 deg,	P =   0.000 deg,	R =    90.000 deg
};
P[6280]{
   GP1:
	UF : 1, UT : 3,		CONFIG : 'N U T, 0, 0, 0',
	X =  25.000  mm,	Y =  124.000  mm,	Z =   15.000 mm,
	W =-180.000 deg,	P =   0.000 deg,	R =    90.000 deg
};
P[6281]{
   GP1:
	UF : 1, UT : 3,		CONFIG : 'N U T, 0, 0, 0',
	X =  25.000  mm,	Y =  124.000  mm,	Z =   -1.000 mm,
	W =-180.000 deg,	P =   0.000 deg,	R =    90.000 deg
};
P[6282]{
   GP1:
	UF : 1, UT : 3,		CONFIG : 'N U T, 0, 0, 0',
	X =  25.000  mm,	Y =  124.000  mm,	Z =   15.000 mm,
	W =-180.000 deg,	P =   0.000 deg,	R =    90.000 deg
};
P[6325]{
   GP1:
	UF : 1, UT : 3,		CONFIG : 'N U T, 0, 0, 0',
	X =  112.000  mm,	Y =  124.000  mm,	Z =   15.000 mm,
	W =-180.000 deg,	P =   0.000 deg,	R =    90.000 deg
};
P[6326]{
   GP1:
	UF : 1, UT : 3,		CONFIG : 'N U T, 0, 0, 0',
	X =  112.000  mm,	Y =  124.000  mm,	Z =   -1.000 mm,
	W =-180.000 deg,	P =   0.000 deg,	R =    90.000 deg
};
P[6327]{
   GP1:
	UF : 1, UT : 3,		CONFIG : 'N U T, 0, 0, 0',
	X =  112.000  mm,	Y =  124.000  mm,	Z =   15.000 mm,
	W =-180.000 deg,	P =   0.000 deg,	R =    90.000 deg
};
P[6376]{
   GP1:
	UF : 1, UT : 3,		CONFIG : 'N U T, 0, 0, 0',
	X =  178.000  mm,	Y =  124.000  mm,	Z =   15.000 mm,
	W =-180.000 deg,	P =   0.000 deg,	R =    90.000 deg
};
P[6377]{
   GP1:
	UF : 1, UT : 3,		CONFIG : 'N U T, 0, 0, 0',
	X =  178.000  mm,	Y =  124.000  mm,	Z =   -1.000 mm,
	W =-180.000 deg,	P =   0.000 deg,	R =    90.000 deg
};
P[6378]{
   GP1:
	UF : 1, UT : 3,		CONFIG : 'N U T, 0, 0, 0',
	X =  178.000  mm,	Y =  124.000  mm,	Z =   15.000 mm,
	W =-180.000 deg,	P =   0.000 deg,	R =    90.000 deg
};
P[6496]{
   GP1:
	UF : 1, UT : 3,		CONFIG : 'N U T, 0, 0, 0',
	X =  7.000  mm,	Y =  130.000  mm,	Z =   15.000 mm,
	W =-180.000 deg,	P =   0.000 deg,	R =    90.000 deg
};
P[6497]{
   GP1:
	UF : 1, UT : 3,		CONFIG : 'N U T, 0, 0, 0',
	X =  7.000  mm,	Y =  130.000  mm,	Z =   -1.000 mm,
	W =-180.000 deg,	P =   0.000 deg,	R =    90.000 deg
};
P[6498]{
   GP1:
	UF : 1, UT : 3,		CONFIG : 'N U T, 0, 0, 0',
	X =  7.000  mm,	Y =  130.000  mm,	Z =   15.000 mm,
	W =-180.000 deg,	P =   0.000 deg,	R =    90.000 deg
};
P[6601]{
   GP1:
	UF : 1, UT : 3,		CONFIG : 'N U T, 0, 0, 0',
	X =  157.000  mm,	Y =  130.000  mm,	Z =   15.000 mm,
	W =-180.000 deg,	P =   0.000 deg,	R =    90.000 deg
};
P[6602]{
   GP1:
	UF : 1, UT : 3,		CONFIG : 'N U T, 0, 0, 0',
